LIN {X -0.033,Y -434.325,Z 655.091,A 0.000,B 0.000,C 90.000,E1 52.316} C_DIS
LIN {X -0.057,Y -434.303,Z 655.091,A 0.000,B 0.000,C 90.000,E1 52.316} C_DIS
LIN {X 0.127,Y -431.665,Z 655.083,A 0.000,B 0.000,C 90.000,E1 50.884} C_DIS
LIN {X 0.114,Y -427.591,Z 655.074,A 0.000,B 0.000,C 90.000,E1 49.218} C_DIS
LIN {X -0.216,Y -420.194,Z 655.054,A 0.000,B 0.000,C 90.000,E1 45.729} C_DIS
LIN {X -0.185,Y -420.290,Z 655.044,A 0.000,B 0.000,C 90.000,E1 44.028} C_DIS
LIN {X 0.050,Y -420.496,Z 655.033,A 0.000,B 0.000,C 90.000,E1 41.962} C_DIS
LIN {X 0.067,Y -421.322,Z 655.016,A 0.000,B 0.000,C 90.000,E1 38.910} C_DIS
LIN {X 0.145,Y -422.879,Z 654.997,A 0.000,B 0.000,C 90.000,E1 35.518} C_DIS
LIN {X 0.123,Y -423.713,Z 654.988,A 0.000,B 0.000,C 90.000,E1 33.833} C_DIS
LIN {X 0.233,Y -424.563,Z 654.979,A 0.000,B 0.000,C 90.000,E1 32.133} C_DIS
LIN {X 0.121,Y -425.591,Z 654.968,A 0.000,B 0.000,C 90.000,E1 30.129} C_DIS
LIN {X -0.166,Y -426.462,Z 654.958,A 0.000,B 0.000,C 90.000,E1 28.487} C_DIS
LIN {X 0.108,Y -427.566,Z 654.947,A 0.000,B 0.000,C 90.000,E1 26.437} C_DIS
LIN {X -0.129,Y -428.218,Z 654.941,A 0.000,B 0.000,C 90.000,E1 25.463} C_DIS
LIN {X 0.186,Y -430.765,Z 654.923,A 0.000,B 0.000,C 90.000,E1 22.078} C_DIS
LIN {X -0.161,Y -431.922,Z 654.915,A 0.000,B 0.000,C 90.000,E1 20.791} C_DIS
LIN {X -0.084,Y -432.910,Z 654.908,A 0.000,B 0.000,C 90.000,E1 19.450} C_DIS
LIN {X 0.100,Y -433.906,Z 654.899,A 0.000,B 0.000,C 90.000,E1 17.764} C_DIS
LIN {X -0.113,Y -434.974,Z 654.890,A 0.000,B 0.000,C 90.000,E1 16.134} C_DIS
LIN {X -0.194,Y -436.724,Z 654.877,A 0.000,B 0.000,C 90.000,E1 13.828} C_DIS
LIN {X -0.037,Y -438.454,Z 654.866,A 0.000,B 0.000,C 90.000,E1 11.827} C_DIS
LIN {X -0.141,Y -440.993,Z 654.851,A 0.000,B 0.000,C 90.000,E1 9.208} C_DIS
LIN {X 0.147,Y -443.830,Z 654.837,A 0.000,B 0.000,C 90.000,E1 6.549} C_DIS
LIN {X 0.026,Y -446.972,Z 654.822,A 0.000,B 0.000,C 90.000,E1 3.955} C_DIS
LIN {X 0.025,Y -449.568,Z 654.811,A 0.000,B 0.000,C 90.000,E1 2.007} C_DIS
LIN {X 0.058,Y -453.757,Z 654.795,A 0.000,B 0.000,C 90.000,E1 359.141} C_DIS
LIN {X 0.221,Y -456.932,Z 654.785,A 0.000,B 0.000,C 90.000,E1 357.192} C_DIS
LIN {X -0.208,Y -460.784,Z 654.772,A 0.000,B 0.000,C 90.000,E1 355.008} C_DIS
LIN {X 0.195,Y -463.089,Z 654.765,A 0.000,B 0.000,C 90.000,E1 353.685} C_DIS
LIN {X -0.239,Y -466.510,Z 654.755,A 0.000,B 0.000,C 90.000,E1 351.837} C_DIS
LIN {X 0.113,Y -469.285,Z 654.746,A 0.000,B 0.000,C 90.000,E1 350.218} C_DIS
LIN {X -0.153,Y -471.492,Z 654.739,A 0.000,B 0.000,C 90.000,E1 348.993} C_DIS
LIN {X -0.164,Y -474.778,Z 654.728,A 0.000,B 0.000,C 90.000,E1 347.117} C_DIS
LIN {X 0.015,Y -478.271,Z 654.718,A 0.000,B 0.000,C 90.000,E1 345.227} C_DIS
LIN {X 0.109,Y -480.603,Z 654.711,A 0.000,B 0.000,C 90.000,E1 343.976} C_DIS
LIN {X 0.084,Y -484.163,Z 654.701,A 0.000,B 0.000,C 90.000,E1 342.127} C_DIS
LIN {X -0.035,Y -487.158,Z 654.692,A 0.000,B 0.000,C 90.000,E1 340.604} C_DIS
LIN {X -0.094,Y -490.244,Z 654.684,A 0.000,B 0.000,C 90.000,E1 339.082} C_DIS
LIN {X 0.079,Y -493.203,Z 654.675,A 0.000,B 0.000,C 90.000,E1 337.539} C_DIS
LIN {X -0.199,Y -495.417,Z 654.669,A 0.000,B 0.000,C 90.000,E1 336.357} C_DIS
LIN {X 0.207,Y -497.465,Z 654.662,A 0.000,B 0.000,C 90.000,E1 335.101} C_DIS
LIN {X -0.139,Y -500.502,Z 654.652,A 0.000,B 0.000,C 90.000,E1 333.332} C_DIS
LIN {X -0.046,Y -504.909,Z 654.638,A 0.000,B 0.000,C 90.000,E1 330.923} C_DIS
LIN {X 0.206,Y -507.111,Z 654.633,A 0.000,B 0.000,C 90.000,E1 329.999} C_DIS
LIN {X 0.155,Y -509.021,Z 654.630,A 0.000,B 0.000,C 90.000,E1 329.410} C_DIS
LIN {X 0.046,Y -510.413,Z 654.629,A 0.000,B 0.000,C 90.000,E1 329.125} C_DIS
LIN {X 0.203,Y -513.157,Z 654.626,A 0.000,B 0.000,C 90.000,E1 328.663} C_DIS
LIN {X 0.021,Y -514.198,Z 654.625,A 0.000,B 0.000,C 90.000,E1 328.535} C_DIS
LIN {X 0.150,Y -515.794,Z 654.624,A 0.000,B 0.000,C 90.000,E1 328.329} C_DIS
LIN {X 0.072,Y -520.333,Z 654.622,A 0.000,B 0.000,C 90.000,E1 327.916} C_DIS
LIN {X -0.043,Y -524.730,Z 654.620,A 0.000,B 0.000,C 90.000,E1 327.533} C_DIS
LIN {X -0.043,Y -530.397,Z 654.617,A 0.000,B 0.000,C 90.000,E1 327.089} C_DIS
LIN {X 0.127,Y -537.887,Z 654.614,A 0.000,B 0.000,C 90.000,E1 326.501} C_DIS
LIN {X -0.157,Y -549.360,Z 654.609,A 0.000,B 0.000,C 90.000,E1 325.595} C_DIS
LIN {X -0.014,Y -554.965,Z 654.606,A 0.000,B 0.000,C 90.000,E1 325.102} C_DIS
LIN {X 0.066,Y -563.274,Z 654.602,A 0.000,B 0.000,C 90.000,E1 324.356} C_DIS
LIN {X 0.115,Y -572.552,Z 654.597,A 0.000,B 0.000,C 90.000,E1 323.497} C_DIS
LIN {X -0.045,Y -581.777,Z 654.592,A 0.000,B 0.000,C 90.000,E1 322.637} C_DIS
LIN {X 0.170,Y -590.747,Z 654.588,A 0.000,B 0.000,C 90.000,E1 321.743} C_DIS
LIN {X 0.239,Y -600.993,Z 654.582,A 0.000,B 0.000,C 90.000,E1 320.723} C_DIS
LIN {X -0.099,Y -606.973,Z 654.578,A 0.000,B 0.000,C 90.000,E1 320.114} C_DIS
LIN {X -0.086,Y -612.730,Z 654.575,A 0.000,B 0.000,C 90.000,E1 319.461} C_DIS
LIN {X 0.197,Y -614.929,Z 654.573,A 0.000,B 0.000,C 90.000,E1 319.175} C_DIS
LIN {X 0.155,Y -619.853,Z 654.570,A 0.000,B 0.000,C 90.000,E1 318.566} C_DIS
LIN {X -0.154,Y -623.691,Z 654.567,A 0.000,B 0.000,C 90.000,E1 318.081} C_DIS
LIN {X -0.226,Y -630.914,Z 654.561,A 0.000,B 0.000,C 90.000,E1 317.067} C_DIS
LIN {X 0.045,Y -633.534,Z 654.559,A 0.000,B 0.000,C 90.000,E1 316.662} C_DIS
LIN {X 0.106,Y -640.171,Z 654.554,A 0.000,B 0.000,C 90.000,E1 315.648} C_DIS
LIN {X 0.282,Y -645.772,Z 654.549,A 0.000,B 0.000,C 90.000,E1 314.757} C_DIS
LIN {X 0.019,Y -652.541,Z 654.543,A 0.000,B 0.000,C 90.000,E1 313.662} C_DIS
LIN {X -0.143,Y -658.239,Z 654.537,A 0.000,B 0.000,C 90.000,E1 312.690} C_DIS
LIN {X -0.214,Y -662.767,Z 654.532,A 0.000,B 0.000,C 90.000,E1 311.838} C_DIS
LIN {X -0.237,Y -667.097,Z 654.528,A 0.000,B 0.000,C 90.000,E1 310.987} C_DIS
LIN {X -0.180,Y -671.728,Z 654.522,A 0.000,B 0.000,C 90.000,E1 310.011} C_DIS
LIN {X -0.078,Y -674.785,Z 654.518,A 0.000,B 0.000,C 90.000,E1 309.277} C_DIS
LIN {X 0.060,Y -677.581,Z 654.514,A 0.000,B 0.000,C 90.000,E1 308.543} C_DIS
LIN {X 0.224,Y -680.153,Z 654.510,A 0.000,B 0.000,C 90.000,E1 307.810} C_DIS
LIN {X 0.023,Y -683.292,Z 654.505,A 0.000,B 0.000,C 90.000,E1 306.870} C_DIS
LIN {X -0.169,Y -685.471,Z 654.501,A 0.000,B 0.000,C 90.000,E1 306.171} C_DIS
LIN {X -0.118,Y -688.806,Z 654.494,A 0.000,B 0.000,C 90.000,E1 304.978} C_DIS
LIN {X 0.344,Y -691.293,Z 654.489,A 0.000,B 0.000,C 90.000,E1 303.992} C_DIS
LIN {X -0.129,Y -693.536,Z 654.484,A 0.000,B 0.000,C 90.000,E1 303.086} C_DIS
LIN {X 0.003,Y -695.668,Z 654.479,A 0.000,B 0.000,C 90.000,E1 302.133} C_DIS
LIN {X -0.204,Y -697.619,Z 654.473,A 0.000,B 0.000,C 90.000,E1 301.209} C_DIS
LIN {X -0.024,Y -699.348,Z 654.468,A 0.000,B 0.000,C 90.000,E1 300.256} C_DIS
LIN {X 0.086,Y -701.210,Z 654.462,A 0.000,B 0.000,C 90.000,E1 299.077} C_DIS
LIN {X 0.292,Y -702.183,Z 654.458,A 0.000,B 0.000,C 90.000,E1 298.359} C_DIS
LIN {X 0.122,Y -703.675,Z 654.451,A 0.000,B 0.000,C 90.000,E1 297.206} C_DIS
LIN {X 0.004,Y -704.754,Z 654.446,A 0.000,B 0.000,C 90.000,E1 296.283} C_DIS
LIN {X -0.076,Y -704.994,Z 654.442,A 0.000,B 0.000,C 90.000,E1 295.591} C_DIS
LIN {X -0.437,Y -704.321,Z 654.440,A 0.000,B 0.000,C 90.000,E1 295.155} C_DIS
LIN {X -0.151,Y -703.852,Z 654.438,A 0.000,B 0.000,C 90.000,E1 294.899} C_DIS
LIN {X -0.008,Y -703.310,Z 654.438,A 0.000,B 0.000,C 90.000,E1 294.771} C_DIS
LIN {X -0.376,Y -700.448,Z 654.435,A 0.000,B 0.000,C 90.000,E1 294.335} C_DIS
LIN {X -0.238,Y -699.553,Z 654.434,A 0.000,B 0.000,C 90.000,E1 294.207} C_DIS
LIN {X -0.103,Y -698.220,Z 654.434,A 0.000,B 0.000,C 90.000,E1 294.079} C_DIS
LIN {X -0.394,Y -694.498,Z 654.433,A 0.000,B 0.000,C 90.000,E1 293.898} C_DIS
LIN {X 0.118,Y -690.985,Z 654.432,A 0.000,B 0.000,C 90.000,E1 293.695} C_DIS
LIN {X -0.140,Y -689.032,Z 654.431,A 0.000,B 0.000,C 90.000,E1 293.643} C_DIS
LIN {X 0.050,Y -681.862,Z 654.430,A 0.000,B 0.000,C 90.000,E1 293.462} C_DIS
LIN {X -0.125,Y -679.782,Z 654.430,A 0.000,B 0.000,C 90.000,E1 293.439} C_DIS
LIN {X -0.175,Y -669.975,Z 654.430,A 0.000,B 0.000,C 90.000,E1 293.334} C_DIS
LIN {X -0.128,Y -662.993,Z 654.429,A 0.000,B 0.000,C 90.000,E1 293.259} C_DIS
LIN {X 0.325,Y -652.595,Z 654.428,A 0.000,B 0.000,C 90.000,E1 293.078} C_DIS
LIN {X -0.159,Y -642.877,Z 654.427,A 0.000,B 0.000,C 90.000,E1 292.950} C_DIS
LIN {X 0.122,Y -629.510,Z 654.426,A 0.000,B 0.000,C 90.000,E1 292.642} C_DIS
LIN {X -0.263,Y -616.266,Z 654.424,A 0.000,B 0.000,C 90.000,E1 292.333} C_DIS
LIN {X -0.196,Y -595.968,Z 654.421,A 0.000,B 0.000,C 90.000,E1 291.716} C_DIS
LIN {X -0.091,Y -578.430,Z 654.418,A 0.000,B 0.000,C 90.000,E1 291.153} C_DIS
LIN {X -0.036,Y -564.068,Z 654.415,A 0.000,B 0.000,C 90.000,E1 290.737} C_DIS
LIN {X 0.221,Y -561.514,Z 654.415,A 0.000,B 0.000,C 90.000,E1 290.610} C_DIS
LIN {X -0.242,Y -559.361,Z 654.414,A 0.000,B 0.000,C 90.000,E1 290.556} C_DIS
LIN {X 0.074,Y -556.501,Z 654.413,A 0.000,B 0.000,C 90.000,E1 290.355} C_DIS
LIN {X 0.019,Y -556.445,Z 654.413,A 0.000,B 0.000,C 90.000,E1 290.355} C_DIS
LIN {X 0.127,Y -555.648,Z 654.412,A 0.000,B 0.000,C 90.000,E1 290.194} C_DIS
LIN {X 0.000,Y -555.094,Z 654.409,A 0.000,B 0.000,C 90.000,E1 289.685} C_DIS
LIN {X 0.116,Y -554.826,Z 654.400,A 0.000,B 0.000,C 90.000,E1 288.000} C_DIS
LIN {X 0.228,Y -554.405,Z 654.391,A 0.000,B 0.000,C 90.000,E1 286.315} C_DIS
LIN {X -0.097,Y -553.844,Z 654.383,A 0.000,B 0.000,C 90.000,E1 284.954} C_DIS
LIN {X 0.110,Y -553.179,Z 654.375,A 0.000,B 0.000,C 90.000,E1 283.536} C_DIS
LIN {X 0.299,Y -552.403,Z 654.368,A 0.000,B 0.000,C 90.000,E1 282.119} C_DIS
LIN {X -0.061,Y -551.460,Z 654.357,A 0.000,B 0.000,C 90.000,E1 280.197} C_DIS
LIN {X -0.120,Y -551.001,Z 654.349,A 0.000,B 0.000,C 90.000,E1 278.803} C_DIS
LIN {X -0.016,Y -550.364,Z 654.336,A 0.000,B 0.000,C 90.000,E1 276.549} C_DIS
LIN {X -0.038,Y -549.996,Z 654.326,A 0.000,B 0.000,C 90.000,E1 274.588} C_DIS
LIN {X -0.219,Y -549.723,Z 654.316,A 0.000,B 0.000,C 90.000,E1 272.922} C_DIS
LIN {X 0.115,Y -549.183,Z 654.307,A 0.000,B 0.000,C 90.000,E1 271.203} C_DIS
LIN {X -0.173,Y -548.544,Z 654.299,A 0.000,B 0.000,C 90.000,E1 269.828} C_DIS
LIN {X 0.137,Y -547.639,Z 654.290,A 0.000,B 0.000,C 90.000,E1 268.108} C_DIS
LIN {X -0.158,Y -546.914,Z 654.282,A 0.000,B 0.000,C 90.000,E1 266.731} C_DIS
LIN {X 0.068,Y -546.038,Z 654.274,A 0.000,B 0.000,C 90.000,E1 265.298} C_DIS
LIN {X -0.178,Y -544.953,Z 654.266,A 0.000,B 0.000,C 90.000,E1 263.913} C_DIS
LIN {X 0.026,Y -543.929,Z 654.260,A 0.000,B 0.000,C 90.000,E1 262.761} C_DIS
LIN {X -0.255,Y -542.397,Z 654.252,A 0.000,B 0.000,C 90.000,E1 261.376} C_DIS
LIN {X -0.109,Y -539.644,Z 654.236,A 0.000,B 0.000,C 90.000,E1 258.522} C_DIS
LIN {X -0.029,Y -537.903,Z 654.225,A 0.000,B 0.000,C 90.000,E1 256.520} C_DIS
LIN {X -0.302,Y -536.949,Z 654.219,A 0.000,B 0.000,C 90.000,E1 255.408} C_DIS
LIN {X 0.198,Y -535.974,Z 654.212,A 0.000,B 0.000,C 90.000,E1 254.212} C_DIS
LIN {X -0.053,Y -533.985,Z 654.201,A 0.000,B 0.000,C 90.000,E1 252.236} C_DIS
LIN {X -0.103,Y -532.964,Z 654.195,A 0.000,B 0.000,C 90.000,E1 251.094} C_DIS
LIN {X 0.003,Y -531.661,Z 654.189,A 0.000,B 0.000,C 90.000,E1 249.934} C_DIS
LIN {X 0.093,Y -530.115,Z 654.182,A 0.000,B 0.000,C 90.000,E1 248.773} C_DIS
LIN {X 0.024,Y -527.580,Z 654.173,A 0.000,B 0.000,C 90.000,E1 247.050} C_DIS
LIN {X -0.241,Y -525.710,Z 654.166,A 0.000,B 0.000,C 90.000,E1 245.921} C_DIS
LIN {X 0.164,Y -523.592,Z 654.160,A 0.000,B 0.000,C 90.000,E1 244.717} C_DIS
LIN {X 0.215,Y -520.776,Z 654.152,A 0.000,B 0.000,C 90.000,E1 243.256} C_DIS
LIN {X -0.013,Y -517.758,Z 654.143,A 0.000,B 0.000,C 90.000,E1 241.820} C_DIS
LIN {X 0.160,Y -514.647,Z 654.135,A 0.000,B 0.000,C 90.000,E1 240.333} C_DIS
LIN {X 0.073,Y -511.274,Z 654.127,A 0.000,B 0.000,C 90.000,E1 238.869} C_DIS
LIN {X -0.181,Y -507.275,Z 654.117,A 0.000,B 0.000,C 90.000,E1 237.120} C_DIS
LIN {X 0.249,Y -504.480,Z 654.111,A 0.000,B 0.000,C 90.000,E1 235.881} C_DIS
LIN {X 0.103,Y -500.618,Z 654.102,A 0.000,B 0.000,C 90.000,E1 234.402} C_DIS
LIN {X -0.245,Y -495.933,Z 654.092,A 0.000,B 0.000,C 90.000,E1 232.637} C_DIS
LIN {X -0.095,Y -491.568,Z 654.082,A 0.000,B 0.000,C 90.000,E1 230.803} C_DIS
LIN {X 0.240,Y -485.807,Z 654.069,A 0.000,B 0.000,C 90.000,E1 228.324} C_DIS
LIN {X -0.065,Y -482.147,Z 654.060,A 0.000,B 0.000,C 90.000,E1 226.824} C_DIS
LIN {X 0.123,Y -479.203,Z 654.053,A 0.000,B 0.000,C 90.000,E1 225.567} C_DIS
LIN {X 0.140,Y -474.764,Z 654.043,A 0.000,B 0.000,C 90.000,E1 223.704} C_DIS
LIN {X -0.078,Y -469.069,Z 654.029,A 0.000,B 0.000,C 90.000,E1 221.229} C_DIS
LIN {X -0.174,Y -464.346,Z 654.017,A 0.000,B 0.000,C 90.000,E1 219.036} C_DIS
LIN {X -0.109,Y -461.027,Z 654.008,A 0.000,B 0.000,C 90.000,E1 217.443} C_DIS
LIN {X -0.003,Y -457.259,Z 653.997,A 0.000,B 0.000,C 90.000,E1 215.518} C_DIS
LIN {X 0.025,Y -454.278,Z 653.988,A 0.000,B 0.000,C 90.000,E1 213.913} C_DIS
LIN {X -0.082,Y -450.089,Z 653.976,A 0.000,B 0.000,C 90.000,E1 211.671} C_DIS
LIN {X -0.068,Y -447.168,Z 653.967,A 0.000,B 0.000,C 90.000,E1 210.050} C_DIS
LIN {X -0.016,Y -444.845,Z 653.960,A 0.000,B 0.000,C 90.000,E1 208.743} C_DIS
LIN {X -0.110,Y -441.283,Z 653.949,A 0.000,B 0.000,C 90.000,E1 206.796} C_DIS
LIN {X -0.095,Y -437.713,Z 653.938,A 0.000,B 0.000,C 90.000,E1 204.823} C_DIS
LIN {X 0.051,Y -434.722,Z 653.929,A 0.000,B 0.000,C 90.000,E1 203.153} C_DIS
LIN {X 0.125,Y -431.154,Z 653.918,A 0.000,B 0.000,C 90.000,E1 201.153} C_DIS
LIN {X -0.144,Y -427.095,Z 653.905,A 0.000,B 0.000,C 90.000,E1 198.852} C_DIS
LIN {X 0.103,Y -423.702,Z 653.893,A 0.000,B 0.000,C 90.000,E1 196.804} C_DIS
LIN {X 0.140,Y -420.426,Z 653.882,A 0.000,B 0.000,C 90.000,E1 194.773} C_DIS
LIN {X -0.115,Y -417.157,Z 653.871,A 0.000,B 0.000,C 90.000,E1 192.771} C_DIS
LIN {X 0.041,Y -412.955,Z 653.856,A 0.000,B 0.000,C 90.000,E1 190.018} C_DIS
LIN {X 0.191,Y -410.923,Z 653.848,A 0.000,B 0.000,C 90.000,E1 188.624} C_DIS
LIN {X -0.145,Y -407.386,Z 653.835,A 0.000,B 0.000,C 90.000,E1 186.258} C_DIS
LIN {X 0.144,Y -403.295,Z 653.817,A 0.000,B 0.000,C 90.000,E1 183.094} C_DIS
LIN {X -0.197,Y -399.883,Z 653.800,A 0.000,B 0.000,C 90.000,E1 180.000} C_DIS
LIN {X 0.169,Y -397.355,Z 653.782,A 0.000,B 0.000,C 90.000,E1 176.788} C_DIS
LIN {X 0.128,Y -395.783,Z 653.767,A 0.000,B 0.000,C 90.000,E1 173.976} C_DIS
LIN {X -0.122,Y -394.947,Z 653.755,A 0.000,B 0.000,C 90.000,E1 171.894} C_DIS
LIN {X -0.008,Y -394.356,Z 653.739,A 0.000,B 0.000,C 90.000,E1 169.050} C_DIS
LIN {X -0.112,Y -394.120,Z 653.721,A 0.000,B 0.000,C 90.000,E1 165.880} C_DIS
LIN {X 0.066,Y -394.291,Z 653.708,A 0.000,B 0.000,C 90.000,E1 163.378} C_DIS
LIN {X -0.012,Y -394.613,Z 653.694,A 0.000,B 0.000,C 90.000,E1 160.913} C_DIS
LIN {X -0.145,Y -394.848,Z 653.686,A 0.000,B 0.000,C 90.000,E1 159.518} C_DIS
LIN {X -0.183,Y -395.390,Z 653.672,A 0.000,B 0.000,C 90.000,E1 157.050} C_DIS
LIN {X 0.105,Y -395.907,Z 653.659,A 0.000,B 0.000,C 90.000,E1 154.537} C_DIS
LIN {X 0.178,Y -396.364,Z 653.647,A 0.000,B 0.000,C 90.000,E1 152.410} C_DIS
LIN {X -0.088,Y -396.937,Z 653.635,A 0.000,B 0.000,C 90.000,E1 150.333} C_DIS
LIN {X -0.079,Y -397.589,Z 653.621,A 0.000,B 0.000,C 90.000,E1 147.867} C_DIS
LIN {X 0.067,Y -398.195,Z 653.612,A 0.000,B 0.000,C 90.000,E1 146.087} C_DIS
LIN {X 0.104,Y -399.261,Z 653.598,A 0.000,B 0.000,C 90.000,E1 143.623} C_DIS
LIN {X -0.024,Y -400.225,Z 653.586,A 0.000,B 0.000,C 90.000,E1 141.537} C_DIS
LIN {X -0.079,Y -401.455,Z 653.573,A 0.000,B 0.000,C 90.000,E1 139.094} C_DIS
LIN {X 0.002,Y -402.564,Z 653.561,A 0.000,B 0.000,C 90.000,E1 136.986} C_DIS
LIN {X -0.006,Y -403.502,Z 653.551,A 0.000,B 0.000,C 90.000,E1 135.243} C_DIS
LIN {X -0.096,Y -405.540,Z 653.534,A 0.000,B 0.000,C 90.000,E1 132.123} C_DIS
LIN {X 0.089,Y -406.483,Z 653.529,A 0.000,B 0.000,C 90.000,E1 131.229} C_DIS
LIN {X 0.148,Y -407.602,Z 653.526,A 0.000,B 0.000,C 90.000,E1 130.701} C_DIS
LIN {X -0.018,Y -408.392,Z 653.524,A 0.000,B 0.000,C 90.000,E1 130.378} C_DIS
LIN {X 0.216,Y -409.094,Z 653.523,A 0.000,B 0.000,C 90.000,E1 130.172} C_DIS
LIN {X 0.059,Y -410.453,Z 653.521,A 0.000,B 0.000,C 90.000,E1 129.806} C_DIS
LIN {X -0.131,Y -413.741,Z 653.519,A 0.000,B 0.000,C 90.000,E1 129.358} C_DIS
LIN {X -0.118,Y -416.974,Z 653.517,A 0.000,B 0.000,C 90.000,E1 129.036} C_DIS
LIN {X -0.103,Y -421.967,Z 653.515,A 0.000,B 0.000,C 90.000,E1 128.624} C_DIS
LIN {X 0.194,Y -429.696,Z 653.511,A 0.000,B 0.000,C 90.000,E1 128.016} C_DIS
LIN {X 0.004,Y -436.340,Z 653.509,A 0.000,B 0.000,C 90.000,E1 127.569} C_DIS
LIN {X -0.075,Y -450.921,Z 653.503,A 0.000,B 0.000,C 90.000,E1 126.583} C_DIS
LIN {X -0.164,Y -462.119,Z 653.499,A 0.000,B 0.000,C 90.000,E1 125.804} C_DIS
LIN {X 0.120,Y -468.409,Z 653.496,A 0.000,B 0.000,C 90.000,E1 125.311} C_DIS
LIN {X -0.187,Y -480.823,Z 653.491,A 0.000,B 0.000,C 90.000,E1 124.405} C_DIS
LIN {X -0.091,Y -488.249,Z 653.488,A 0.000,B 0.000,C 90.000,E1 123.785} C_DIS
LIN {X 0.106,Y -496.820,Z 653.484,A 0.000,B 0.000,C 90.000,E1 123.038} C_DIS
LIN {X 0.079,Y -508.137,Z 653.478,A 0.000,B 0.000,C 90.000,E1 122.005} C_DIS
LIN {X -0.090,Y -514.962,Z 653.474,A 0.000,B 0.000,C 90.000,E1 121.386} C_DIS
LIN {X -0.114,Y -521.788,Z 653.471,A 0.000,B 0.000,C 90.000,E1 120.718} C_DIS
LIN {X 0.241,Y -526.990,Z 653.468,A 0.000,B 0.000,C 90.000,E1 120.129} C_DIS
LIN {X 0.090,Y -531.773,Z 653.465,A 0.000,B 0.000,C 90.000,E1 119.617} C_DIS
LIN {X 0.204,Y -536.168,Z 653.462,A 0.000,B 0.000,C 90.000,E1 119.077} C_DIS
LIN {X -0.125,Y -540.425,Z 653.459,A 0.000,B 0.000,C 90.000,E1 118.565} C_DIS
LIN {X -0.004,Y -544.201,Z 653.456,A 0.000,B 0.000,C 90.000,E1 118.025} C_DIS
LIN {X -0.154,Y -548.668,Z 653.452,A 0.000,B 0.000,C 90.000,E1 117.334} C_DIS
LIN {X -0.009,Y -552.514,Z 653.448,A 0.000,B 0.000,C 90.000,E1 116.616} C_DIS
LIN {X -0.074,Y -556.096,Z 653.444,A 0.000,B 0.000,C 90.000,E1 115.924} C_DIS
LIN {X 0.132,Y -559.198,Z 653.440,A 0.000,B 0.000,C 90.000,E1 115.207} C_DIS
LIN {X -0.180,Y -563.754,Z 653.434,A 0.000,B 0.000,C 90.000,E1 114.131} C_DIS
LIN {X 0.269,Y -566.998,Z 653.429,A 0.000,B 0.000,C 90.000,E1 113.259} C_DIS
LIN {X 0.015,Y -569.930,Z 653.425,A 0.000,B 0.000,C 90.000,E1 112.461} C_DIS
LIN {X 0.006,Y -572.587,Z 653.420,A 0.000,B 0.000,C 90.000,E1 111.642} C_DIS
LIN {X -0.193,Y -574.998,Z 653.416,A 0.000,B 0.000,C 90.000,E1 110.844} C_DIS
LIN {X 0.187,Y -578.411,Z 653.408,A 0.000,B 0.000,C 90.000,E1 109.450} C_DIS
LIN {X -0.140,Y -580.338,Z 653.404,A 0.000,B 0.000,C 90.000,E1 108.671} C_DIS
LIN {X -0.215,Y -583.227,Z 653.396,A 0.000,B 0.000,C 90.000,E1 107.330} C_DIS
LIN {X -0.197,Y -586.668,Z 653.387,A 0.000,B 0.000,C 90.000,E1 105.717} C_DIS
LIN {X 0.259,Y -591.327,Z 653.375,A 0.000,B 0.000,C 90.000,E1 103.536} C_DIS
LIN {X -0.116,Y -594.164,Z 653.368,A 0.000,B 0.000,C 90.000,E1 102.243} C_DIS
LIN {X 0.135,Y -596.935,Z 653.361,A 0.000,B 0.000,C 90.000,E1 100.894} C_DIS
LIN {X 0.029,Y -600.214,Z 653.352,A 0.000,B 0.000,C 90.000,E1 99.321} C_DIS
LIN {X 0.177,Y -602.813,Z 653.345,A 0.000,B 0.000,C 90.000,E1 97.992} C_DIS
LIN {X 0.139,Y -604.673,Z 653.339,A 0.000,B 0.000,C 90.000,E1 96.947} C_DIS
LIN {X 0.044,Y -606.484,Z 653.333,A 0.000,B 0.000,C 90.000,E1 95.910} C_DIS
LIN {X -0.107,Y -608.829,Z 653.324,A 0.000,B 0.000,C 90.000,E1 94.359} C_DIS
LIN {X 0.120,Y -610.679,Z 653.317,A 0.000,B 0.000,C 90.000,E1 93.037} C_DIS
LIN {X 0.014,Y -612.361,Z 653.308,A 0.000,B 0.000,C 90.000,E1 91.489} C_DIS
LIN {X -0.046,Y -613.252,Z 653.303,A 0.000,B 0.000,C 90.000,E1 90.458} C_DIS
LIN {X 0.227,Y -613.795,Z 653.298,A 0.000,B 0.000,C 90.000,E1 89.656} C_DIS
LIN {X 0.188,Y -614.324,Z 653.292,A 0.000,B 0.000,C 90.000,E1 88.625} C_DIS
LIN {X 0.170,Y -614.625,Z 653.287,A 0.000,B 0.000,C 90.000,E1 87.593} C_DIS
LIN {X -0.134,Y -614.758,Z 653.282,A 0.000,B 0.000,C 90.000,E1 86.846} C_DIS
LIN {X -0.138,Y -614.715,Z 653.277,A 0.000,B 0.000,C 90.000,E1 85.812} C_DIS
LIN {X 0.195,Y -614.350,Z 653.270,A 0.000,B 0.000,C 90.000,E1 84.489} C_DIS
LIN {X 0.167,Y -613.909,Z 653.264,A 0.000,B 0.000,C 90.000,E1 83.457} C_DIS
LIN {X 0.270,Y -613.340,Z 653.258,A 0.000,B 0.000,C 90.000,E1 82.413} C_DIS
LIN {X -0.319,Y -612.541,Z 653.252,A 0.000,B 0.000,C 90.000,E1 81.432} C_DIS
LIN {X -0.130,Y -610.777,Z 653.244,A 0.000,B 0.000,C 90.000,E1 79.859} C_DIS
LIN {X 0.282,Y -609.078,Z 653.236,A 0.000,B 0.000,C 90.000,E1 78.522} C_DIS
LIN {X 0.186,Y -607.161,Z 653.229,A 0.000,B 0.000,C 90.000,E1 77.229} C_DIS
LIN {X 0.058,Y -605.085,Z 653.222,A 0.000,B 0.000,C 90.000,E1 75.936} C_DIS
LIN {X 0.041,Y -602.779,Z 653.215,A 0.000,B 0.000,C 90.000,E1 74.629} C_DIS
LIN {X -0.017,Y -600.306,Z 653.207,A 0.000,B 0.000,C 90.000,E1 73.323} C_DIS
LIN {X 0.051,Y -597.637,Z 653.200,A 0.000,B 0.000,C 90.000,E1 72.000} C_DIS
LIN {X -0.189,Y -595.247,Z 653.194,A 0.000,B 0.000,C 90.000,E1 70.967} C_DIS
LIN {X 0.099,Y -592.668,Z 653.188,A 0.000,B 0.000,C 90.000,E1 69.880} C_DIS
LIN {X 0.111,Y -590.521,Z 653.184,A 0.000,B 0.000,C 90.000,E1 69.082} C_DIS
LIN {X 0.102,Y -588.176,Z 653.179,A 0.000,B 0.000,C 90.000,E1 68.284} C_DIS
LIN {X 0.066,Y -585.603,Z 653.175,A 0.000,B 0.000,C 90.000,E1 67.486} C_DIS
LIN {X -0.181,Y -583.795,Z 653.172,A 0.000,B 0.000,C 90.000,E1 66.975} C_DIS
LIN {X 0.129,Y -579.675,Z 653.166,A 0.000,B 0.000,C 90.000,E1 65.869} C_DIS
LIN {X 0.082,Y -575.434,Z 653.160,A 0.000,B 0.000,C 90.000,E1 64.793} C_DIS
LIN {X -0.221,Y -573.115,Z 653.157,A 0.000,B 0.000,C 90.000,E1 64.280} C_DIS
LIN {X 0.067,Y -569.505,Z 653.153,A 0.000,B 0.000,C 90.000,E1 63.435} C_DIS
LIN {X 0.051,Y -565.533,Z 653.148,A 0.000,B 0.000,C 90.000,E1 62.615} C_DIS
LIN {X -0.225,Y -563.352,Z 653.146,A 0.000,B 0.000,C 90.000,E1 62.231} C_DIS
LIN {X 0.150,Y -560.300,Z 653.143,A 0.000,B 0.000,C 90.000,E1 61.641} C_DIS
LIN {X 0.033,Y -556.114,Z 653.139,A 0.000,B 0.000,C 90.000,E1 60.973} C_DIS
LIN {X -0.252,Y -551.407,Z 653.135,A 0.000,B 0.000,C 90.000,E1 60.333} C_DIS
LIN {X -0.099,Y -547.510,Z 653.132,A 0.000,B 0.000,C 90.000,E1 59.793} C_DIS
LIN {X 0.156,Y -542.722,Z 653.129,A 0.000,B 0.000,C 90.000,E1 59.203} C_DIS
LIN {X 0.064,Y -537.484,Z 653.126,A 0.000,B 0.000,C 90.000,E1 58.663} C_DIS
LIN {X -0.043,Y -532.338,Z 653.123,A 0.000,B 0.000,C 90.000,E1 58.201} C_DIS
LIN {X -0.165,Y -528.302,Z 653.121,A 0.000,B 0.000,C 90.000,E1 57.867} C_DIS
LIN {X 0.048,Y -521.880,Z 653.119,A 0.000,B 0.000,C 90.000,E1 57.375} C_DIS
LIN {X 0.118,Y -517.021,Z 653.117,A 0.000,B 0.000,C 90.000,E1 57.041} C_DIS
LIN {X 0.238,Y -510.328,Z 653.115,A 0.000,B 0.000,C 90.000,E1 56.628} C_DIS
LIN {X -0.149,Y -503.595,Z 653.113,A 0.000,B 0.000,C 90.000,E1 56.294} C_DIS
LIN {X -0.111,Y -496.760,Z 653.111,A 0.000,B 0.000,C 90.000,E1 55.928} C_DIS
LIN {X 0.055,Y -476.690,Z 653.105,A 0.000,B 0.000,C 90.000,E1 54.848} C_DIS
LIN {X -0.035,Y -450.032,Z 653.097,A 0.000,B 0.000,C 90.000,E1 53.417} C_DIS
LIN {X 0.155,Y -435.467,Z 653.092,A 0.000,B 0.000,C 90.000,E1 52.557} C_DIS
LIN {X -0.154,Y -434.792,Z 653.092,A 0.000,B 0.000,C 90.000,E1 52.557} C_DIS
LIN {X -0.178,Y -434.753,Z 653.092,A 0.000,B 0.000,C 90.000,E1 52.557} C_DIS
LIN {X -0.037,Y -431.278,Z 653.082,A 0.000,B 0.000,C 90.000,E1 50.723} C_DIS
LIN {X -0.034,Y -422.090,Z 653.059,A 0.000,B 0.000,C 90.000,E1 46.701} C_DIS
LIN {X -0.237,Y -420.789,Z 653.056,A 0.000,B 0.000,C 90.000,E1 46.053} C_DIS
LIN {X 0.011,Y -420.605,Z 653.055,A 0.000,B 0.000,C 90.000,E1 45.850} C_DIS
LIN {X -0.179,Y -420.784,Z 653.046,A 0.000,B 0.000,C 90.000,E1 44.352} C_DIS
LIN {X 0.071,Y -420.990,Z 653.035,A 0.000,B 0.000,C 90.000,E1 42.285} C_DIS
LIN {X -0.214,Y -421.769,Z 653.018,A 0.000,B 0.000,C 90.000,E1 39.277} C_DIS
LIN {X 0.048,Y -422.906,Z 653.003,A 0.000,B 0.000,C 90.000,E1 36.537} C_DIS
LIN {X 0.100,Y -423.467,Z 652.997,A 0.000,B 0.000,C 90.000,E1 35.518} C_DIS
LIN {X -0.122,Y -424.148,Z 652.990,A 0.000,B 0.000,C 90.000,E1 34.199} C_DIS
LIN {X 0.211,Y -425.135,Z 652.979,A 0.000,B 0.000,C 90.000,E1 32.133} C_DIS
LIN {X 0.113,Y -426.134,Z 652.968,A 0.000,B 0.000,C 90.000,E1 30.129} C_DIS
LIN {X -0.165,Y -426.998,Z 652.958,A 0.000,B 0.000,C 90.000,E1 28.487} C_DIS
LIN {X 0.109,Y -428.328,Z 652.945,A 0.000,B 0.000,C 90.000,E1 26.104} C_DIS
LIN {X 0.041,Y -430.633,Z 652.927,A 0.000,B 0.000,C 90.000,E1 22.770} C_DIS
LIN {X 0.070,Y -432.079,Z 652.917,A 0.000,B 0.000,C 90.000,E1 21.099} C_DIS
LIN {X -0.031,Y -433.303,Z 652.908,A 0.000,B 0.000,C 90.000,E1 19.450} C_DIS
LIN {X -0.020,Y -434.482,Z 652.897,A 0.000,B 0.000,C 90.000,E1 17.457} C_DIS
LIN {X -0.115,Y -435.781,Z 652.886,A 0.000,B 0.000,C 90.000,E1 15.481} C_DIS
LIN {X -0.037,Y -437.903,Z 652.871,A 0.000,B 0.000,C 90.000,E1 12.827} C_DIS
LIN {X 0.057,Y -439.621,Z 652.860,A 0.000,B 0.000,C 90.000,E1 10.838} C_DIS
LIN {X 0.112,Y -441.575,Z 652.849,A 0.000,B 0.000,C 90.000,E1 8.859} C_DIS
LIN {X -0.189,Y -444.080,Z 652.837,A 0.000,B 0.000,C 90.000,E1 6.606} C_DIS
LIN {X -0.028,Y -446.747,Z 652.824,A 0.000,B 0.000,C 90.000,E1 4.302} C_DIS
LIN {X 0.143,Y -448.452,Z 652.817,A 0.000,B 0.000,C 90.000,E1 2.980} C_DIS
LIN {X 0.049,Y -452.022,Z 652.802,A 0.000,B 0.000,C 90.000,E1 0.401} C_DIS
LIN {X -0.135,Y -455.995,Z 652.788,A 0.000,B 0.000,C 90.000,E1 357.879} C_DIS
LIN {X -0.160,Y -459.789,Z 652.776,A 0.000,B 0.000,C 90.000,E1 355.641} C_DIS
LIN {X -0.038,Y -462.638,Z 652.767,A 0.000,B 0.000,C 90.000,E1 354.033} C_DIS
LIN {X 0.239,Y -465.457,Z 652.758,A 0.000,B 0.000,C 90.000,E1 352.413} C_DIS
LIN {X -0.153,Y -467.743,Z 652.751,A 0.000,B 0.000,C 90.000,E1 351.197} C_DIS
LIN {X 0.042,Y -471.058,Z 652.741,A 0.000,B 0.000,C 90.000,E1 349.285} C_DIS
LIN {X -0.145,Y -474.852,Z 652.728,A 0.000,B 0.000,C 90.000,E1 347.117} C_DIS
LIN {X -0.123,Y -478.951,Z 652.716,A 0.000,B 0.000,C 90.000,E1 344.936} C_DIS
LIN {X -0.190,Y -482.428,Z 652.706,A 0.000,B 0.000,C 90.000,E1 343.087} C_DIS
LIN {X -0.034,Y -486.043,Z 652.696,A 0.000,B 0.000,C 90.000,E1 341.221} C_DIS
LIN {X -0.067,Y -490.306,Z 652.684,A 0.000,B 0.000,C 90.000,E1 339.082} C_DIS
LIN {X 0.107,Y -493.257,Z 652.675,A 0.000,B 0.000,C 90.000,E1 337.539} C_DIS
LIN {X -0.171,Y -495.444,Z 652.669,A 0.000,B 0.000,C 90.000,E1 336.357} C_DIS
LIN {X 0.236,Y -497.488,Z 652.662,A 0.000,B 0.000,C 90.000,E1 335.101} C_DIS
LIN {X -0.110,Y -500.496,Z 652.652,A 0.000,B 0.000,C 90.000,E1 333.332} C_DIS
LIN {X 0.294,Y -505.432,Z 652.637,A 0.000,B 0.000,C 90.000,E1 330.589} C_DIS
LIN {X -0.141,Y -507.593,Z 652.632,A 0.000,B 0.000,C 90.000,E1 329.744} C_DIS
LIN {X 0.070,Y -509.547,Z 652.629,A 0.000,B 0.000,C 90.000,E1 329.125} C_DIS
LIN {X -0.014,Y -511.062,Z 652.627,A 0.000,B 0.000,C 90.000,E1 328.791} C_DIS
LIN {X -0.030,Y -513.017,Z 652.625,A 0.000,B 0.000,C 90.000,E1 328.456} C_DIS
LIN {X 0.044,Y -515.238,Z 652.623,A 0.000,B 0.000,C 90.000,E1 328.152} C_DIS
LIN {X 0.139,Y -516.431,Z 652.622,A 0.000,B 0.000,C 90.000,E1 327.995} C_DIS
LIN {X 0.064,Y -520.438,Z 652.620,A 0.000,B 0.000,C 90.000,E1 327.612} C_DIS
LIN {X -0.133,Y -525.746,Z 652.618,A 0.000,B 0.000,C 90.000,E1 327.168} C_DIS
LIN {X 0.026,Y -535.818,Z 652.613,A 0.000,B 0.000,C 90.000,E1 326.373} C_DIS
LIN {X -0.264,Y -547.461,Z 652.608,A 0.000,B 0.000,C 90.000,E1 325.468} C_DIS
LIN {X -0.090,Y -554.513,Z 652.605,A 0.000,B 0.000,C 90.000,E1 324.848} C_DIS
LIN {X -0.077,Y -562.894,Z 652.601,A 0.000,B 0.000,C 90.000,E1 324.116} C_DIS
LIN {X -0.067,Y -569.664,Z 652.597,A 0.000,B 0.000,C 90.000,E1 323.497} C_DIS
LIN {X 0.200,Y -580.237,Z 652.592,A 0.000,B 0.000,C 90.000,E1 322.477} C_DIS
LIN {X 0.064,Y -589.288,Z 652.587,A 0.000,B 0.000,C 90.000,E1 321.618} C_DIS
LIN {X -0.293,Y -600.894,Z 652.581,A 0.000,B 0.000,C 90.000,E1 320.517} C_DIS
LIN {X 0.201,Y -606.934,Z 652.577,A 0.000,B 0.000,C 90.000,E1 319.828} C_DIS
LIN {X -0.253,Y -612.740,Z 652.573,A 0.000,B 0.000,C 90.000,E1 319.218} C_DIS
LIN {X -0.202,Y -618.156,Z 652.570,A 0.000,B 0.000,C 90.000,E1 318.566} C_DIS
LIN {X -0.059,Y -622.125,Z 652.567,A 0.000,B 0.000,C 90.000,E1 318.038} C_DIS
LIN {X 0.270,Y -629.486,Z 652.561,A 0.000,B 0.000,C 90.000,E1 316.986} C_DIS
LIN {X 0.033,Y -632.998,Z 652.558,A 0.000,B 0.000,C 90.000,E1 316.500} C_DIS
LIN {X 0.085,Y -639.716,Z 652.553,A 0.000,B 0.000,C 90.000,E1 315.486} C_DIS
LIN {X 0.256,Y -645.340,Z 652.548,A 0.000,B 0.000,C 90.000,E1 314.595} C_DIS
LIN {X 0.194,Y -651.382,Z 652.542,A 0.000,B 0.000,C 90.000,E1 313.623} C_DIS
LIN {X -0.255,Y -657.147,Z 652.537,A 0.000,B 0.000,C 90.000,E1 312.690} C_DIS
LIN {X -0.339,Y -661.769,Z 652.532,A 0.000,B 0.000,C 90.000,E1 311.838} C_DIS
LIN {X 0.104,Y -665.633,Z 652.528,A 0.000,B 0.000,C 90.000,E1 311.067} C_DIS
LIN {X 0.145,Y -670.346,Z 652.523,A 0.000,B 0.000,C 90.000,E1 310.092} C_DIS
LIN {X 0.238,Y -673.570,Z 652.519,A 0.000,B 0.000,C 90.000,E1 309.358} C_DIS
LIN {X -0.164,Y -676.467,Z 652.515,A 0.000,B 0.000,C 90.000,E1 308.669} C_DIS
LIN {X -0.015,Y -679.113,Z 652.511,A 0.000,B 0.000,C 90.000,E1 307.935} C_DIS
LIN {X 0.311,Y -682.308,Z 652.505,A 0.000,B 0.000,C 90.000,E1 306.950} C_DIS
LIN {X 0.111,Y -684.558,Z 652.501,A 0.000,B 0.000,C 90.000,E1 306.251} C_DIS
LIN {X 0.177,Y -688.656,Z 652.494,A 0.000,B 0.000,C 90.000,E1 304.818} C_DIS
LIN {X -0.326,Y -691.141,Z 652.488,A 0.000,B 0.000,C 90.000,E1 303.913} C_DIS
LIN {X 0.003,Y -693.981,Z 652.482,A 0.000,B 0.000,C 90.000,E1 302.704} C_DIS
LIN {X -0.201,Y -696.621,Z 652.475,A 0.000,B 0.000,C 90.000,E1 301.544} C_DIS
LIN {X -0.032,Y -698.479,Z 652.470,A 0.000,B 0.000,C 90.000,E1 300.590} C_DIS
LIN {X -0.200,Y -700.127,Z 652.465,A 0.000,B 0.000,C 90.000,E1 299.667} C_DIS
LIN {X 0.267,Y -701.647,Z 652.460,A 0.000,B 0.000,C 90.000,E1 298.693} C_DIS
LIN {X 0.416,Y -703.232,Z 652.453,A 0.000,B 0.000,C 90.000,E1 297.513} C_DIS
LIN {X 0.263,Y -704.647,Z 652.447,A 0.000,B 0.000,C 90.000,E1 296.360} C_DIS
LIN {X -0.083,Y -704.861,Z 652.445,A 0.000,B 0.000,C 90.000,E1 296.155} C_DIS
LIN {X 0.185,Y -704.999,Z 652.443,A 0.000,B 0.000,C 90.000,E1 295.668} C_DIS
LIN {X -0.162,Y -704.829,Z 652.441,A 0.000,B 0.000,C 90.000,E1 295.463} C_DIS
LIN {X 0.114,Y -704.106,Z 652.439,A 0.000,B 0.000,C 90.000,E1 294.975} C_DIS
LIN {X -0.238,Y -703.189,Z 652.438,A 0.000,B 0.000,C 90.000,E1 294.771} C_DIS
LIN {X 0.321,Y -700.318,Z 652.435,A 0.000,B 0.000,C 90.000,E1 294.259} C_DIS
LIN {X 0.171,Y -699.364,Z 652.434,A 0.000,B 0.000,C 90.000,E1 294.155} C_DIS
LIN {X -0.332,Y -697.936,Z 652.434,A 0.000,B 0.000,C 90.000,E1 294.079} C_DIS
LIN {X -0.074,Y -695.897,Z 652.433,A 0.000,B 0.000,C 90.000,E1 293.951} C_DIS
LIN {X -0.044,Y -690.251,Z 652.432,A 0.000,B 0.000,C 90.000,E1 293.695} C_DIS
LIN {X -0.262,Y -688.188,Z 652.431,A 0.000,B 0.000,C 90.000,E1 293.643} C_DIS
LIN {X 0.088,Y -681.443,Z 652.430,A 0.000,B 0.000,C 90.000,E1 293.462} C_DIS
LIN {X -0.217,Y -673.441,Z 652.430,A 0.000,B 0.000,C 90.000,E1 293.387} C_DIS
LIN {X 0.131,Y -663.519,Z 652.429,A 0.000,B 0.000,C 90.000,E1 293.259} C_DIS
LIN {X 0.078,Y -653.615,Z 652.429,A 0.000,B 0.000,C 90.000,E1 293.131} C_DIS
LIN {X 0.221,Y -643.660,Z 652.428,A 0.000,B 0.000,C 90.000,E1 292.950} C_DIS
LIN {X -0.046,Y -630.294,Z 652.426,A 0.000,B 0.000,C 90.000,E1 292.695} C_DIS
LIN {X -0.212,Y -620.523,Z 652.425,A 0.000,B 0.000,C 90.000,E1 292.461} C_DIS
LIN {X -0.185,Y -603.676,Z 652.422,A 0.000,B 0.000,C 90.000,E1 291.972} C_DIS
LIN {X 0.135,Y -582.740,Z 652.418,A 0.000,B 0.000,C 90.000,E1 291.280} C_DIS
LIN {X -0.243,Y -575.451,Z 652.417,A 0.000,B 0.000,C 90.000,E1 291.099} C_DIS
LIN {X -0.109,Y -563.481,Z 652.415,A 0.000,B 0.000,C 90.000,E1 290.737} C_DIS
LIN {X -0.062,Y -560.523,Z 652.414,A 0.000,B 0.000,C 90.000,E1 290.610} C_DIS
LIN {X 0.009,Y -556.596,Z 652.413,A 0.000,B 0.000,C 90.000,E1 290.375} C_DIS
LIN {X -0.047,Y -556.537,Z 652.413,A 0.000,B 0.000,C 90.000,E1 290.375} C_DIS
LIN {X -0.322,Y -555.710,Z 652.412,A 0.000,B 0.000,C 90.000,E1 290.248} C_DIS
LIN {X 0.073,Y -555.187,Z 652.409,A 0.000,B 0.000,C 90.000,E1 289.685} C_DIS
LIN {X 0.191,Y -554.933,Z 652.400,A 0.000,B 0.000,C 90.000,E1 288.000} C_DIS
LIN {X 0.305,Y -554.500,Z 652.391,A 0.000,B 0.000,C 90.000,E1 286.315} C_DIS
LIN {X -0.018,Y -553.954,Z 652.383,A 0.000,B 0.000,C 90.000,E1 284.954} C_DIS
LIN {X 0.192,Y -553.290,Z 652.375,A 0.000,B 0.000,C 90.000,E1 283.536} C_DIS
LIN {X -0.039,Y -552.366,Z 652.366,A 0.000,B 0.000,C 90.000,E1 281.883} C_DIS
LIN {X -0.173,Y -551.287,Z 652.352,A 0.000,B 0.000,C 90.000,E1 279.378} C_DIS
LIN {X -0.071,Y -550.605,Z 652.340,A 0.000,B 0.000,C 90.000,E1 277.125} C_DIS
LIN {X -0.131,Y -550.203,Z 652.330,A 0.000,B 0.000,C 90.000,E1 275.448} C_DIS
LIN {X 0.191,Y -549.961,Z 652.322,A 0.000,B 0.000,C 90.000,E1 274.012} C_DIS
LIN {X -0.125,Y -549.758,Z 652.316,A 0.000,B 0.000,C 90.000,E1 272.922} C_DIS
LIN {X 0.207,Y -549.245,Z 652.307,A 0.000,B 0.000,C 90.000,E1 271.203} C_DIS
LIN {X -0.079,Y -548.604,Z 652.299,A 0.000,B 0.000,C 90.000,E1 269.828} C_DIS
LIN {X -0.267,Y -547.573,Z 652.288,A 0.000,B 0.000,C 90.000,E1 267.879} C_DIS
LIN {X -0.020,Y -546.827,Z 652.280,A 0.000,B 0.000,C 90.000,E1 266.445} C_DIS
LIN {X 0.166,Y -546.139,Z 652.274,A 0.000,B 0.000,C 90.000,E1 265.298} C_DIS
LIN {X -0.078,Y -545.065,Z 652.266,A 0.000,B 0.000,C 90.000,E1 263.913} C_DIS
LIN {X 0.127,Y -544.061,Z 652.260,A 0.000,B 0.000,C 90.000,E1 262.761} C_DIS
LIN {X -0.152,Y -542.517,Z 652.252,A 0.000,B 0.000,C 90.000,E1 261.376} C_DIS
LIN {X -0.003,Y -539.761,Z 652.236,A 0.000,B 0.000,C 90.000,E1 258.522} C_DIS
LIN {X 0.145,Y -537.784,Z 652.224,A 0.000,B 0.000,C 90.000,E1 256.228} C_DIS
LIN {X 0.112,Y -536.346,Z 652.214,A 0.000,B 0.000,C 90.000,E1 254.519} C_DIS
LIN {X 0.092,Y -535.199,Z 652.208,A 0.000,B 0.000,C 90.000,E1 253.378} C_DIS
LIN {X -0.186,Y -533.321,Z 652.197,A 0.000,B 0.000,C 90.000,E1 251.402} C_DIS
LIN {X -0.272,Y -532.461,Z 652.192,A 0.000,B 0.000,C 90.000,E1 250.550} C_DIS
LIN {X -0.174,Y -531.038,Z 652.185,A 0.000,B 0.000,C 90.000,E1 249.390} C_DIS
LIN {X 0.086,Y -528.943,Z 652.177,A 0.000,B 0.000,C 90.000,E1 247.922} C_DIS
LIN {X 0.144,Y -527.681,Z 652.173,A 0.000,B 0.000,C 90.000,E1 247.050} C_DIS
LIN {X -0.120,Y -525.795,Z 652.166,A 0.000,B 0.000,C 90.000,E1 245.921} C_DIS
LIN {X 0.286,Y -523.672,Z 652.160,A 0.000,B 0.000,C 90.000,E1 244.717} C_DIS
LIN {X -0.127,Y -520.824,Z 652.152,A 0.000,B 0.000,C 90.000,E1 243.307} C_DIS
LIN {X -0.134,Y -517.792,Z 652.144,A 0.000,B 0.000,C 90.000,E1 241.847} C_DIS
LIN {X -0.078,Y -515.358,Z 652.137,A 0.000,B 0.000,C 90.000,E1 240.667} C_DIS
LIN {X -0.151,Y -511.976,Z 652.129,A 0.000,B 0.000,C 90.000,E1 239.203} C_DIS
LIN {X -0.016,Y -508.633,Z 652.121,A 0.000,B 0.000,C 90.000,E1 237.709} C_DIS
LIN {X 0.161,Y -505.874,Z 652.114,A 0.000,B 0.000,C 90.000,E1 236.501} C_DIS
LIN {X -0.048,Y -504.479,Z 652.111,A 0.000,B 0.000,C 90.000,E1 235.928} C_DIS
LIN {X -0.070,Y -501.373,Z 652.104,A 0.000,B 0.000,C 90.000,E1 234.736} C_DIS
LIN {X 0.006,Y -496.681,Z 652.094,A 0.000,B 0.000,C 90.000,E1 232.924} C_DIS
LIN {X 0.022,Y -491.547,Z 652.082,A 0.000,B 0.000,C 90.000,E1 230.803} C_DIS
LIN {X -0.009,Y -485.762,Z 652.069,A 0.000,B 0.000,C 90.000,E1 228.366} C_DIS
LIN {X 0.048,Y -482.108,Z 652.060,A 0.000,B 0.000,C 90.000,E1 226.824} C_DIS
LIN {X 0.234,Y -479.134,Z 652.053,A 0.000,B 0.000,C 90.000,E1 225.567} C_DIS
LIN {X 0.142,Y -475.465,Z 652.045,A 0.000,B 0.000,C 90.000,E1 224.028} C_DIS
LIN {X -0.052,Y -469.723,Z 652.031,A 0.000,B 0.000,C 90.000,E1 221.553} C_DIS
LIN {X -0.070,Y -464.270,Z 652.017,A 0.000,B 0.000,C 90.000,E1 219.036} C_DIS
LIN {X -0.260,Y -460.308,Z 652.006,A 0.000,B 0.000,C 90.000,E1 217.156} C_DIS
LIN {X -0.171,Y -456.556,Z 651.996,A 0.000,B 0.000,C 90.000,E1 215.231} C_DIS
LIN {X 0.220,Y -453.578,Z 651.987,A 0.000,B 0.000,C 90.000,E1 213.579} C_DIS
LIN {X 0.097,Y -449.467,Z 651.974,A 0.000,B 0.000,C 90.000,E1 211.337} C_DIS
LIN {X 0.012,Y -445.446,Z 651.962,A 0.000,B 0.000,C 90.000,E1 209.077} C_DIS
LIN {X -0.064,Y -441.841,Z 651.951,A 0.000,B 0.000,C 90.000,E1 207.129} C_DIS
LIN {X -0.029,Y -438.280,Z 651.940,A 0.000,B 0.000,C 90.000,E1 205.155} C_DIS
LIN {X 0.138,Y -434.657,Z 651.929,A 0.000,B 0.000,C 90.000,E1 203.153} C_DIS
LIN {X 0.055,Y -431.112,Z 651.918,A 0.000,B 0.000,C 90.000,E1 201.173} C_DIS
LIN {X -0.128,Y -427.633,Z 651.907,A 0.000,B 0.000,C 90.000,E1 199.195} C_DIS
LIN {X -0.005,Y -424.245,Z 651.895,A 0.000,B 0.000,C 90.000,E1 197.166} C_DIS
LIN {X 0.222,Y -420.410,Z 651.882,A 0.000,B 0.000,C 90.000,E1 194.773} C_DIS
LIN {X -0.034,Y -417.165,Z 651.871,A 0.000,B 0.000,C 90.000,E1 192.771} C_DIS
LIN {X 0.122,Y -412.978,Z 651.856,A 0.000,B 0.000,C 90.000,E1 190.018} C_DIS
LIN {X -0.135,Y -410.952,Z 651.848,A 0.000,B 0.000,C 90.000,E1 188.681} C_DIS
LIN {X -0.065,Y -407.420,Z 651.835,A 0.000,B 0.000,C 90.000,E1 186.258} C_DIS
LIN {X -0.177,Y -403.340,Z 651.817,A 0.000,B 0.000,C 90.000,E1 183.151} C_DIS
LIN {X -0.114,Y -399.937,Z 651.800,A 0.000,B 0.000,C 90.000,E1 180.000} C_DIS
LIN {X -0.107,Y -397.668,Z 651.784,A 0.000,B 0.000,C 90.000,E1 177.192} C_DIS
LIN {X -0.179,Y -395.869,Z 651.767,A 0.000,B 0.000,C 90.000,E1 174.033} C_DIS
LIN {X -0.034,Y -395.047,Z 651.755,A 0.000,B 0.000,C 90.000,E1 171.894} C_DIS
LIN {X 0.120,Y -394.518,Z 651.741,A 0.000,B 0.000,C 90.000,E1 169.398} C_DIS
LIN {X -0.022,Y -394.264,Z 651.726,A 0.000,B 0.000,C 90.000,E1 166.589} C_DIS
LIN {X 0.102,Y -394.317,Z 651.714,A 0.000,B 0.000,C 90.000,E1 164.448} C_DIS
LIN {X -0.207,Y -394.502,Z 651.704,A 0.000,B 0.000,C 90.000,E1 162.725} C_DIS
LIN {X 0.155,Y -394.850,Z 651.692,A 0.000,B 0.000,C 90.000,E1 160.550} C_DIS
LIN {X 0.225,Y -395.147,Z 651.682,A 0.000,B 0.000,C 90.000,E1 158.773} C_DIS
LIN {X -0.068,Y -395.578,Z 651.672,A 0.000,B 0.000,C 90.000,E1 157.050} C_DIS
LIN {X 0.087,Y -396.221,Z 651.657,A 0.000,B 0.000,C 90.000,E1 154.204} C_DIS
LIN {X -0.012,Y -396.695,Z 651.645,A 0.000,B 0.000,C 90.000,E1 152.103} C_DIS
LIN {X -0.082,Y -397.226,Z 651.633,A 0.000,B 0.000,C 90.000,E1 149.999} C_DIS
LIN {X 0.060,Y -397.811,Z 651.622,A 0.000,B 0.000,C 90.000,E1 147.867} C_DIS
LIN {X -0.121,Y -398.429,Z 651.612,A 0.000,B 0.000,C 90.000,E1 146.135} C_DIS
LIN {X 0.017,Y -399.462,Z 651.598,A 0.000,B 0.000,C 90.000,E1 143.657} C_DIS
LIN {X 0.016,Y -400.282,Z 651.588,A 0.000,B 0.000,C 90.000,E1 141.904} C_DIS
LIN {X -0.155,Y -401.263,Z 651.577,A 0.000,B 0.000,C 90.000,E1 139.828} C_DIS
LIN {X -0.164,Y -402.146,Z 651.567,A 0.000,B 0.000,C 90.000,E1 138.081} C_DIS
LIN {X -0.063,Y -403.227,Z 651.555,A 0.000,B 0.000,C 90.000,E1 135.972} C_DIS
LIN {X 0.222,Y -404.134,Z 651.546,A 0.000,B 0.000,C 90.000,E1 134.190} C_DIS
LIN {X 0.207,Y -405.776,Z 651.532,A 0.000,B 0.000,C 90.000,E1 131.757} C_DIS
LIN {X 0.176,Y -406.547,Z 651.528,A 0.000,B 0.000,C 90.000,E1 131.067} C_DIS
LIN {X 0.150,Y -407.789,Z 651.524,A 0.000,B 0.000,C 90.000,E1 130.378} C_DIS
LIN {X -0.060,Y -409.732,Z 651.521,A 0.000,B 0.000,C 90.000,E1 129.769} C_DIS
LIN {X 0.158,Y -411.311,Z 651.520,A 0.000,B 0.000,C 90.000,E1 129.483} C_DIS
LIN {X -0.183,Y -412.205,Z 651.519,A 0.000,B 0.000,C 90.000,E1 129.358} C_DIS
LIN {X 0.059,Y -413.369,Z 651.518,A 0.000,B 0.000,C 90.000,E1 129.152} C_DIS
LIN {X 0.017,Y -417.503,Z 651.515,A 0.000,B 0.000,C 90.000,E1 128.749} C_DIS
LIN {X -0.151,Y -422.309,Z 651.513,A 0.000,B 0.000,C 90.000,E1 128.382} C_DIS
LIN {X 0.212,Y -433.567,Z 651.509,A 0.000,B 0.000,C 90.000,E1 127.523} C_DIS
LIN {X 0.022,Y -449.811,Z 651.503,A 0.000,B 0.000,C 90.000,E1 126.457} C_DIS
LIN {X -0.098,Y -459.428,Z 651.499,A 0.000,B 0.000,C 90.000,E1 125.804} C_DIS
LIN {X 0.234,Y -465.730,Z 651.496,A 0.000,B 0.000,C 90.000,E1 125.311} C_DIS
LIN {X 0.085,Y -476.451,Z 651.492,A 0.000,B 0.000,C 90.000,E1 124.532} C_DIS
LIN {X 0.030,Y -482.491,Z 651.489,A 0.000,B 0.000,C 90.000,E1 124.072} C_DIS
LIN {X 0.187,Y -486.802,Z 651.487,A 0.000,B 0.000,C 90.000,E1 123.706} C_DIS
LIN {X 0.060,Y -495.422,Z 651.483,A 0.000,B 0.000,C 90.000,E1 123.007} C_DIS
LIN {X -0.100,Y -503.926,Z 651.479,A 0.000,B 0.000,C 90.000,E1 122.260} C_DIS
LIN {X -0.083,Y -512.113,Z 651.475,A 0.000,B 0.000,C 90.000,E1 121.514} C_DIS
LIN {X -0.139,Y -520.548,Z 651.471,A 0.000,B 0.000,C 90.000,E1 120.718} C_DIS
LIN {X -0.047,Y -526.812,Z 651.467,A 0.000,B 0.000,C 90.000,E1 120.050} C_DIS
LIN {X -0.009,Y -530.449,Z 651.465,A 0.000,B 0.000,C 90.000,E1 119.667} C_DIS
LIN {X -0.018,Y -534.889,Z 651.462,A 0.000,B 0.000,C 90.000,E1 119.155} C_DIS
LIN {X -0.071,Y -539.283,Z 651.459,A 0.000,B 0.000,C 90.000,E1 118.615} C_DIS
LIN {X -0.316,Y -544.182,Z 651.455,A 0.000,B 0.000,C 90.000,E1 117.975} C_DIS
LIN {X -0.090,Y -547.897,Z 651.452,A 0.000,B 0.000,C 90.000,E1 117.385} C_DIS
LIN {X -0.070,Y -552.629,Z 651.447,A 0.000,B 0.000,C 90.000,E1 116.539} C_DIS
LIN {X -0.139,Y -556.253,Z 651.444,A 0.000,B 0.000,C 90.000,E1 115.848} C_DIS
LIN {X -0.276,Y -559.975,Z 651.439,A 0.000,B 0.000,C 90.000,E1 115.027} C_DIS
LIN {X -0.062,Y -564.543,Z 651.433,A 0.000,B 0.000,C 90.000,E1 113.898} C_DIS
LIN {X -0.119,Y -567.799,Z 651.428,A 0.000,B 0.000,C 90.000,E1 113.078} C_DIS
LIN {X -0.149,Y -570.709,Z 651.424,A 0.000,B 0.000,C 90.000,E1 112.259} C_DIS
LIN {X 0.166,Y -573.327,Z 651.419,A 0.000,B 0.000,C 90.000,E1 111.408} C_DIS
LIN {X 0.150,Y -574.952,Z 651.416,A 0.000,B 0.000,C 90.000,E1 110.865} C_DIS
LIN {X -0.185,Y -577.820,Z 651.410,A 0.000,B 0.000,C 90.000,E1 109.812} C_DIS
LIN {X -0.136,Y -580.461,Z 651.404,A 0.000,B 0.000,C 90.000,E1 108.725} C_DIS
LIN {X 0.170,Y -583.387,Z 651.397,A 0.000,B 0.000,C 90.000,E1 107.347} C_DIS
LIN {X 0.044,Y -587.429,Z 651.386,A 0.000,B 0.000,C 90.000,E1 105.481} C_DIS
LIN {X 0.260,Y -591.574,Z 651.376,A 0.000,B 0.000,C 90.000,E1 103.592} C_DIS
LIN {X -0.113,Y -594.473,Z 651.368,A 0.000,B 0.000,C 90.000,E1 102.299} C_DIS
LIN {X -0.155,Y -597.832,Z 651.359,A 0.000,B 0.000,C 90.000,E1 100.715} C_DIS
LIN {X 0.039,Y -600.610,Z 651.352,A 0.000,B 0.000,C 90.000,E1 99.378} C_DIS
LIN {X 0.193,Y -603.264,Z 651.345,A 0.000,B 0.000,C 90.000,E1 98.049} C_DIS
LIN {X 0.159,Y -605.185,Z 651.339,A 0.000,B 0.000,C 90.000,E1 97.004} C_DIS
LIN {X -0.281,Y -607.412,Z 651.332,A 0.000,B 0.000,C 90.000,E1 95.739} C_DIS
LIN {X 0.199,Y -609.773,Z 651.323,A 0.000,B 0.000,C 90.000,E1 94.131} C_DIS
LIN {X 0.164,Y -611.242,Z 651.317,A 0.000,B 0.000,C 90.000,E1 93.094} C_DIS
LIN {X -0.239,Y -612.711,Z 651.310,A 0.000,B 0.000,C 90.000,E1 91.835} C_DIS
LIN {X 0.041,Y -613.471,Z 651.306,A 0.000,B 0.000,C 90.000,E1 91.031} C_DIS
LIN {X 0.298,Y -614.468,Z 651.299,A 0.000,B 0.000,C 90.000,E1 89.714} C_DIS
LIN {X 0.267,Y -614.995,Z 651.293,A 0.000,B 0.000,C 90.000,E1 88.682} C_DIS
LIN {X 0.260,Y -615.336,Z 651.287,A 0.000,B 0.000,C 90.000,E1 87.650} C_DIS
LIN {X 0.263,Y -615.461,Z 651.281,A 0.000,B 0.000,C 90.000,E1 86.617} C_DIS
LIN {X -0.055,Y -615.297,Z 651.274,A 0.000,B 0.000,C 90.000,E1 85.355} C_DIS
LIN {X 0.277,Y -614.829,Z 651.267,A 0.000,B 0.000,C 90.000,E1 84.033} C_DIS
LIN {X -0.294,Y -614.326,Z 651.261,A 0.000,B 0.000,C 90.000,E1 83.053} C_DIS
LIN {X -0.180,Y -613.638,Z 651.256,A 0.000,B 0.000,C 90.000,E1 82.008} C_DIS
LIN {X 0.185,Y -612.901,Z 651.251,A 0.000,B 0.000,C 90.000,E1 81.197} C_DIS
LIN {X -0.071,Y -611.408,Z 651.244,A 0.000,B 0.000,C 90.000,E1 79.926} C_DIS
LIN {X -0.136,Y -609.649,Z 651.237,A 0.000,B 0.000,C 90.000,E1 78.634} C_DIS
LIN {X 0.244,Y -607.742,Z 651.230,A 0.000,B 0.000,C 90.000,E1 77.297} C_DIS
LIN {X 0.262,Y -605.608,Z 651.222,A 0.000,B 0.000,C 90.000,E1 75.992} C_DIS
LIN {X -0.215,Y -603.744,Z 651.217,A 0.000,B 0.000,C 90.000,E1 74.991} C_DIS
LIN {X 0.019,Y -601.772,Z 651.211,A 0.000,B 0.000,C 90.000,E1 73.921} C_DIS
LIN {X 0.220,Y -599.680,Z 651.205,A 0.000,B 0.000,C 90.000,E1 72.851} C_DIS
LIN {X -0.002,Y -597.469,Z 651.199,A 0.000,B 0.000,C 90.000,E1 71.819} C_DIS
LIN {X -0.137,Y -595.660,Z 651.195,A 0.000,B 0.000,C 90.000,E1 71.040} C_DIS
LIN {X 0.353,Y -593.046,Z 651.189,A 0.000,B 0.000,C 90.000,E1 69.934} C_DIS
LIN {X 0.048,Y -590.058,Z 651.183,A 0.000,B 0.000,C 90.000,E1 68.901} C_DIS
LIN {X 0.032,Y -587.630,Z 651.178,A 0.000,B 0.000,C 90.000,E1 68.103} C_DIS
LIN {X -0.136,Y -583.990,Z 651.172,A 0.000,B 0.000,C 90.000,E1 67.050} C_DIS
LIN {X -0.122,Y -579.851,Z 651.167,A 0.000,B 0.000,C 90.000,E1 65.973} C_DIS
LIN {X -0.156,Y -575.539,Z 651.161,A 0.000,B 0.000,C 90.000,E1 64.897} C_DIS
LIN {X 0.064,Y -573.221,Z 651.157,A 0.000,B 0.000,C 90.000,E1 64.332} C_DIS
LIN {X 0.099,Y -569.505,Z 651.153,A 0.000,B 0.000,C 90.000,E1 63.512} C_DIS
LIN {X -0.244,Y -566.880,Z 651.150,A 0.000,B 0.000,C 90.000,E1 62.999} C_DIS
LIN {X 0.065,Y -563.299,Z 651.146,A 0.000,B 0.000,C 90.000,E1 62.281} C_DIS
LIN {X 0.076,Y -559.277,Z 651.142,A 0.000,B 0.000,C 90.000,E1 61.591} C_DIS
LIN {X -0.070,Y -555.792,Z 651.139,A 0.000,B 0.000,C 90.000,E1 61.051} C_DIS
LIN {X 0.139,Y -550.756,Z 651.135,A 0.000,B 0.000,C 90.000,E1 60.333} C_DIS
LIN {X 0.069,Y -547.557,Z 651.133,A 0.000,B 0.000,C 90.000,E1 59.921} C_DIS
LIN {X 0.329,Y -542.765,Z 651.130,A 0.000,B 0.000,C 90.000,E1 59.331} C_DIS
LIN {X -0.039,Y -537.465,Z 651.127,A 0.000,B 0.000,C 90.000,E1 58.820} C_DIS
LIN {X 0.007,Y -534.213,Z 651.125,A 0.000,B 0.000,C 90.000,E1 58.535} C_DIS
LIN {X 0.071,Y -532.076,Z 651.124,A 0.000,B 0.000,C 90.000,E1 58.329} C_DIS
LIN {X -0.062,Y -526.238,Z 651.122,A 0.000,B 0.000,C 90.000,E1 57.867} C_DIS
LIN {X 0.069,Y -521.278,Z 651.120,A 0.000,B 0.000,C 90.000,E1 57.502} C_DIS
LIN {X -0.240,Y -514.793,Z 651.117,A 0.000,B 0.000,C 90.000,E1 57.120} C_DIS
LIN {X -0.052,Y -507.965,Z 651.115,A 0.000,B 0.000,C 90.000,E1 56.707} C_DIS
LIN {X 0.297,Y -499.647,Z 651.113,A 0.000,B 0.000,C 90.000,E1 56.215} C_DIS
LIN {X 0.141,Y -479.576,Z 651.107,A 0.000,B 0.000,C 90.000,E1 55.182} C_DIS
LIN {X -0.138,Y -462.730,Z 651.102,A 0.000,B 0.000,C 90.000,E1 54.322} C_DIS
LIN {X 0.075,Y -444.555,Z 651.096,A 0.000,B 0.000,C 90.000,E1 53.290} C_DIS
LIN {X -0.010,Y -435.217,Z 651.093,A 0.000,B 0.000,C 90.000,E1 52.763} C_DIS
LIN {X -0.034,Y -435.210,Z 651.093,A 0.000,B 0.000,C 90.000,E1 52.763} C_DIS
LIN {X 0.097,Y -431.801,Z 651.083,A 0.000,B 0.000,C 90.000,E1 50.964} C_DIS
LIN {X 0.021,Y -431.089,Z 651.081,A 0.000,B 0.000,C 90.000,E1 50.642} C_DIS
LIN {X 0.018,Y -421.944,Z 651.059,A 0.000,B 0.000,C 90.000,E1 46.620} C_DIS
LIN {X -0.110,Y -421.128,Z 651.057,A 0.000,B 0.000,C 90.000,E1 46.215} C_DIS
LIN {X -0.228,Y -421.322,Z 651.044,A 0.000,B 0.000,C 90.000,E1 43.947} C_DIS
LIN {X 0.057,Y -421.834,Z 651.027,A 0.000,B 0.000,C 90.000,E1 40.862} C_DIS
LIN {X 0.087,Y -422.473,Z 651.016,A 0.000,B 0.000,C 90.000,E1 38.830} C_DIS
LIN {X -0.188,Y -423.535,Z 651.003,A 0.000,B 0.000,C 90.000,E1 36.503} C_DIS
LIN {X 0.020,Y -424.622,Z 650.991,A 0.000,B 0.000,C 90.000,E1 34.452} C_DIS
LIN {X 0.129,Y -425.581,Z 650.980,A 0.000,B 0.000,C 90.000,E1 32.418} C_DIS
LIN {X 0.036,Y -426.705,Z 650.967,A 0.000,B 0.000,C 90.000,E1 30.079} C_DIS
LIN {X -0.010,Y -427.392,Z 650.960,A 0.000,B 0.000,C 90.000,E1 28.743} C_DIS
LIN {X -0.097,Y -428.462,Z 650.949,A 0.000,B 0.000,C 90.000,E1 26.744} C_DIS
LIN {X -0.152,Y -429.410,Z 650.939,A 0.000,B 0.000,C 90.000,E1 25.079} C_DIS
LIN {X 0.036,Y -431.144,Z 650.926,A 0.000,B 0.000,C 90.000,E1 22.717} C_DIS
LIN {X 0.080,Y -432.534,Z 650.917,A 0.000,B 0.000,C 90.000,E1 21.046} C_DIS
LIN {X -0.008,Y -433.719,Z 650.908,A 0.000,B 0.000,C 90.000,E1 19.396} C_DIS
LIN {X -0.164,Y -435.096,Z 650.895,A 0.000,B 0.000,C 90.000,E1 17.094} C_DIS
LIN {X -0.125,Y -436.641,Z 650.882,A 0.000,B 0.000,C 90.000,E1 14.773} C_DIS
LIN {X 0.032,Y -438.263,Z 650.871,A 0.000,B 0.000,C 90.000,E1 12.771} C_DIS
LIN {X 0.009,Y -440.613,Z 650.856,A 0.000,B 0.000,C 90.000,E1 10.141} C_DIS
LIN {X -0.089,Y -443.282,Z 650.842,A 0.000,B 0.000,C 90.000,E1 7.530} C_DIS
LIN {X -0.195,Y -445.131,Z 650.833,A 0.000,B 0.000,C 90.000,E1 5.910} C_DIS
LIN {X -0.186,Y -448.733,Z 650.816,A 0.000,B 0.000,C 90.000,E1 2.980} C_DIS
LIN {X 0.000,Y -452.787,Z 650.800,A 0.000,B 0.000,C 90.000,E1 360.000} C_DIS
LIN {X -0.225,Y -457.202,Z 650.785,A 0.000,B 0.000,C 90.000,E1 357.249} C_DIS
LIN {X 0.037,Y -460.473,Z 650.774,A 0.000,B 0.000,C 90.000,E1 355.298} C_DIS
LIN {X 0.003,Y -463.885,Z 650.763,A 0.000,B 0.000,C 90.000,E1 353.394} C_DIS
LIN {X -0.140,Y -467.837,Z 650.751,A 0.000,B 0.000,C 90.000,E1 351.197} C_DIS
LIN {X 0.058,Y -471.126,Z 650.741,A 0.000,B 0.000,C 90.000,E1 349.285} C_DIS
LIN {X 0.040,Y -474.383,Z 650.730,A 0.000,B 0.000,C 90.000,E1 347.409} C_DIS
LIN {X 0.055,Y -478.418,Z 650.718,A 0.000,B 0.000,C 90.000,E1 345.227} C_DIS
LIN {X -0.001,Y -481.309,Z 650.709,A 0.000,B 0.000,C 90.000,E1 343.685} C_DIS
LIN {X 0.132,Y -484.910,Z 650.699,A 0.000,B 0.000,C 90.000,E1 341.819} C_DIS
LIN {X -0.115,Y -488.497,Z 650.689,A 0.000,B 0.000,C 90.000,E1 340.007} C_DIS
LIN {X -0.012,Y -490.961,Z 650.682,A 0.000,B 0.000,C 90.000,E1 338.773} C_DIS
LIN {X 0.134,Y -493.284,Z 650.675,A 0.000,B 0.000,C 90.000,E1 337.539} C_DIS
LIN {X -0.143,Y -495.470,Z 650.669,A 0.000,B 0.000,C 90.000,E1 336.357} C_DIS
LIN {X 0.265,Y -497.488,Z 650.662,A 0.000,B 0.000,C 90.000,E1 335.101} C_DIS
LIN {X -0.081,Y -500.491,Z 650.652,A 0.000,B 0.000,C 90.000,E1 333.332} C_DIS
LIN {X -0.055,Y -505.877,Z 650.635,A 0.000,B 0.000,C 90.000,E1 330.333} C_DIS
LIN {X 0.205,Y -508.088,Z 650.630,A 0.000,B 0.000,C 90.000,E1 329.410} C_DIS
LIN {X -0.278,Y -510.030,Z 650.627,A 0.000,B 0.000,C 90.000,E1 328.869} C_DIS
LIN {X 0.067,Y -511.260,Z 650.625,A 0.000,B 0.000,C 90.000,E1 328.535} C_DIS
LIN {X -0.212,Y -513.816,Z 650.623,A 0.000,B 0.000,C 90.000,E1 328.122} C_DIS
LIN {X 0.137,Y -516.025,Z 650.621,A 0.000,B 0.000,C 90.000,E1 327.788} C_DIS
LIN {X 0.171,Y -520.316,Z 650.619,A 0.000,B 0.000,C 90.000,E1 327.327} C_DIS
LIN {X 0.059,Y -524.100,Z 650.617,A 0.000,B 0.000,C 90.000,E1 326.993} C_DIS
LIN {X 0.103,Y -537.545,Z 650.611,A 0.000,B 0.000,C 90.000,E1 325.928} C_DIS
LIN {X 0.164,Y -547.730,Z 650.606,A 0.000,B 0.000,C 90.000,E1 325.102} C_DIS
LIN {X -0.096,Y -554.800,Z 650.603,A 0.000,B 0.000,C 90.000,E1 324.529} C_DIS
LIN {X -0.365,Y -564.537,Z 650.598,A 0.000,B 0.000,C 90.000,E1 323.703} C_DIS
LIN {X -0.030,Y -571.322,Z 650.595,A 0.000,B 0.000,C 90.000,E1 323.050} C_DIS
LIN {X 0.266,Y -579.329,Z 650.591,A 0.000,B 0.000,C 90.000,E1 322.271} C_DIS
LIN {X 0.025,Y -589.783,Z 650.585,A 0.000,B 0.000,C 90.000,E1 321.295} C_DIS
LIN {X 0.235,Y -600.073,Z 650.579,A 0.000,B 0.000,C 90.000,E1 320.275} C_DIS
LIN {X -0.119,Y -605.824,Z 650.576,A 0.000,B 0.000,C 90.000,E1 319.703} C_DIS
LIN {X 0.035,Y -609.430,Z 650.574,A 0.000,B 0.000,C 90.000,E1 319.299} C_DIS
LIN {X 0.155,Y -613.960,Z 650.571,A 0.000,B 0.000,C 90.000,E1 318.771} C_DIS
LIN {X -0.003,Y -617.134,Z 650.569,A 0.000,B 0.000,C 90.000,E1 318.405} C_DIS
LIN {X 0.054,Y -622.195,Z 650.565,A 0.000,B 0.000,C 90.000,E1 317.757} C_DIS
LIN {X 0.044,Y -628.728,Z 650.560,A 0.000,B 0.000,C 90.000,E1 316.863} C_DIS
LIN {X 0.304,Y -631.412,Z 650.558,A 0.000,B 0.000,C 90.000,E1 316.458} C_DIS
LIN {X -0.124,Y -638.274,Z 650.553,A 0.000,B 0.000,C 90.000,E1 315.486} C_DIS
LIN {X 0.026,Y -644.023,Z 650.548,A 0.000,B 0.000,C 90.000,E1 314.595} C_DIS
LIN {X -0.084,Y -650.916,Z 650.542,A 0.000,B 0.000,C 90.000,E1 313.500} C_DIS
LIN {X -0.011,Y -653.901,Z 650.539,A 0.000,B 0.000,C 90.000,E1 313.014} C_DIS
LIN {X -0.097,Y -656.798,Z 650.536,A 0.000,B 0.000,C 90.000,E1 312.528} C_DIS
LIN {X 0.295,Y -660.874,Z 650.532,A 0.000,B 0.000,C 90.000,E1 311.757} C_DIS
LIN {X -0.207,Y -664.807,Z 650.528,A 0.000,B 0.000,C 90.000,E1 311.067} C_DIS
LIN {X -0.204,Y -667.890,Z 650.525,A 0.000,B 0.000,C 90.000,E1 310.458} C_DIS
LIN {X -0.139,Y -671.276,Z 650.521,A 0.000,B 0.000,C 90.000,E1 309.725} C_DIS
LIN {X -0.036,Y -674.372,Z 650.517,A 0.000,B 0.000,C 90.000,E1 308.991} C_DIS
LIN {X 0.098,Y -677.215,Z 650.513,A 0.000,B 0.000,C 90.000,E1 308.257} C_DIS
LIN {X 0.261,Y -679.769,Z 650.509,A 0.000,B 0.000,C 90.000,E1 307.523} C_DIS
LIN {X 0.054,Y -682.908,Z 650.503,A 0.000,B 0.000,C 90.000,E1 306.583} C_DIS
LIN {X -0.141,Y -685.075,Z 650.499,A 0.000,B 0.000,C 90.000,E1 305.884} C_DIS
LIN {X -0.096,Y -688.533,Z 650.493,A 0.000,B 0.000,C 90.000,E1 304.692} C_DIS
LIN {X 0.358,Y -691.023,Z 650.487,A 0.000,B 0.000,C 90.000,E1 303.706} C_DIS
LIN {X 0.105,Y -693.938,Z 650.481,A 0.000,B 0.000,C 90.000,E1 302.546} C_DIS
LIN {X -0.108,Y -696.584,Z 650.474,A 0.000,B 0.000,C 90.000,E1 301.386} C_DIS
LIN {X 0.043,Y -698.005,Z 650.470,A 0.000,B 0.000,C 90.000,E1 300.669} C_DIS
LIN {X 0.139,Y -700.147,Z 650.464,A 0.000,B 0.000,C 90.000,E1 299.489} C_DIS
LIN {X -0.001,Y -701.699,Z 650.459,A 0.000,B 0.000,C 90.000,E1 298.565} C_DIS
LIN {X 0.149,Y -703.359,Z 650.452,A 0.000,B 0.000,C 90.000,E1 297.385} C_DIS
LIN {X -0.004,Y -704.774,Z 650.446,A 0.000,B 0.000,C 90.000,E1 296.232} C_DIS
LIN {X -0.081,Y -704.901,Z 650.442,A 0.000,B 0.000,C 90.000,E1 295.540} C_DIS
LIN {X -0.142,Y -704.157,Z 650.439,A 0.000,B 0.000,C 90.000,E1 295.079} C_DIS
LIN {X 0.143,Y -703.534,Z 650.438,A 0.000,B 0.000,C 90.000,E1 294.823} C_DIS
LIN {X -0.226,Y -700.696,Z 650.435,A 0.000,B 0.000,C 90.000,E1 294.387} C_DIS
LIN {X -0.089,Y -699.907,Z 650.435,A 0.000,B 0.000,C 90.000,E1 294.259} C_DIS
LIN {X 0.046,Y -698.819,Z 650.434,A 0.000,B 0.000,C 90.000,E1 294.131} C_DIS
LIN {X -0.105,Y -697.159,Z 650.433,A 0.000,B 0.000,C 90.000,E1 294.027} C_DIS
LIN {X -0.240,Y -691.327,Z 650.432,A 0.000,B 0.000,C 90.000,E1 293.770} C_DIS
LIN {X -0.200,Y -689.378,Z 650.432,A 0.000,B 0.000,C 90.000,E1 293.695} C_DIS
LIN {X 0.193,Y -686.969,Z 650.431,A 0.000,B 0.000,C 90.000,E1 293.590} C_DIS
LIN {X 0.004,Y -680.222,Z 650.430,A 0.000,B 0.000,C 90.000,E1 293.462} C_DIS
LIN {X 0.276,Y -670.501,Z 650.430,A 0.000,B 0.000,C 90.000,E1 293.334} C_DIS
LIN {X 0.018,Y -661.453,Z 650.429,A 0.000,B 0.000,C 90.000,E1 293.259} C_DIS
LIN {X -0.155,Y -651.284,Z 650.428,A 0.000,B 0.000,C 90.000,E1 293.131} C_DIS
LIN {X -0.045,Y -641.684,Z 650.428,A 0.000,B 0.000,C 90.000,E1 292.950} C_DIS
LIN {X 0.194,Y -631.487,Z 650.426,A 0.000,B 0.000,C 90.000,E1 292.717} C_DIS
LIN {X 0.178,Y -618.491,Z 650.424,A 0.000,B 0.000,C 90.000,E1 292.386} C_DIS
LIN {X 0.261,Y -597.994,Z 650.421,A 0.000,B 0.000,C 90.000,E1 291.770} C_DIS
LIN {X 0.161,Y -580.571,Z 650.418,A 0.000,B 0.000,C 90.000,E1 291.227} C_DIS
LIN {X -0.212,Y -573.103,Z 650.417,A 0.000,B 0.000,C 90.000,E1 291.046} C_DIS
LIN {X -0.152,Y -563.051,Z 650.415,A 0.000,B 0.000,C 90.000,E1 290.737} C_DIS
LIN {X 0.194,Y -559.718,Z 650.414,A 0.000,B 0.000,C 90.000,E1 290.556} C_DIS
LIN {X 0.010,Y -556.544,Z 650.413,A 0.000,B 0.000,C 90.000,E1 290.375} C_DIS
LIN {X -0.045,Y -556.502,Z 650.413,A 0.000,B 0.000,C 90.000,E1 290.375} C_DIS
LIN {X 0.070,Y -555.911,Z 650.413,A 0.000,B 0.000,C 90.000,E1 290.248} C_DIS
LIN {X -0.196,Y -555.570,Z 650.411,A 0.000,B 0.000,C 90.000,E1 290.066} C_DIS
LIN {X 0.093,Y -555.242,Z 650.410,A 0.000,B 0.000,C 90.000,E1 289.758} C_DIS
LIN {X -0.105,Y -555.032,Z 650.401,A 0.000,B 0.000,C 90.000,E1 288.109} C_DIS
LIN {X 0.259,Y -554.719,Z 650.393,A 0.000,B 0.000,C 90.000,E1 286.677} C_DIS
LIN {X -0.178,Y -554.343,Z 650.387,A 0.000,B 0.000,C 90.000,E1 285.607} C_DIS
LIN {X 0.039,Y -553.729,Z 650.379,A 0.000,B 0.000,C 90.000,E1 284.189} C_DIS
LIN {X 0.123,Y -553.115,Z 650.373,A 0.000,B 0.000,C 90.000,E1 283.063} C_DIS
LIN {X -0.108,Y -552.113,Z 650.362,A 0.000,B 0.000,C 90.000,E1 281.130} C_DIS
LIN {X 0.077,Y -551.308,Z 650.351,A 0.000,B 0.000,C 90.000,E1 279.151} C_DIS
LIN {X 0.154,Y -550.710,Z 650.340,A 0.000,B 0.000,C 90.000,E1 277.182} C_DIS
LIN {X 0.042,Y -550.292,Z 650.331,A 0.000,B 0.000,C 90.000,E1 275.511} C_DIS
LIN {X -0.172,Y -550.011,Z 650.323,A 0.000,B 0.000,C 90.000,E1 274.131} C_DIS
LIN {X 0.152,Y -549.724,Z 650.315,A 0.000,B 0.000,C 90.000,E1 272.694} C_DIS
LIN {X -0.115,Y -549.307,Z 650.307,A 0.000,B 0.000,C 90.000,E1 271.318} C_DIS
LIN {X 0.200,Y -548.554,Z 650.298,A 0.000,B 0.000,C 90.000,E1 269.599} C_DIS
LIN {X 0.009,Y -547.530,Z 650.287,A 0.000,B 0.000,C 90.000,E1 267.650} C_DIS
LIN {X 0.251,Y -546.803,Z 650.279,A 0.000,B 0.000,C 90.000,E1 266.216} C_DIS
LIN {X -0.065,Y -546.063,Z 650.273,A 0.000,B 0.000,C 90.000,E1 265.122} C_DIS
LIN {X 0.183,Y -545.012,Z 650.265,A 0.000,B 0.000,C 90.000,E1 263.685} C_DIS
LIN {X -0.159,Y -543.972,Z 650.259,A 0.000,B 0.000,C 90.000,E1 262.591} C_DIS
LIN {X 0.175,Y -542.402,Z 650.251,A 0.000,B 0.000,C 90.000,E1 261.141} C_DIS
LIN {X -0.201,Y -539.687,Z 650.235,A 0.000,B 0.000,C 90.000,E1 258.342} C_DIS
LIN {X -0.048,Y -537.728,Z 650.223,A 0.000,B 0.000,C 90.000,E1 256.047} C_DIS
LIN {X -0.079,Y -536.240,Z 650.213,A 0.000,B 0.000,C 90.000,E1 254.338} C_DIS
LIN {X 0.142,Y -534.575,Z 650.203,A 0.000,B 0.000,C 90.000,E1 252.598} C_DIS
LIN {X -0.180,Y -532.978,Z 650.194,A 0.000,B 0.000,C 90.000,E1 250.913} C_DIS
LIN {X -0.268,Y -531.998,Z 650.189,A 0.000,B 0.000,C 90.000,E1 250.061} C_DIS
LIN {X -0.176,Y -530.431,Z 650.183,A 0.000,B 0.000,C 90.000,E1 248.901} C_DIS
LIN {X 0.270,Y -528.345,Z 650.175,A 0.000,B 0.000,C 90.000,E1 247.411} C_DIS
LIN {X -0.192,Y -526.513,Z 650.168,A 0.000,B 0.000,C 90.000,E1 246.305} C_DIS
LIN {X -0.090,Y -523.898,Z 650.160,A 0.000,B 0.000,C 90.000,E1 244.845} C_DIS
LIN {X 0.288,Y -521.599,Z 650.154,A 0.000,B 0.000,C 90.000,E1 243.640} C_DIS
LIN {X 0.159,Y -519.207,Z 650.147,A 0.000,B 0.000,C 90.000,E1 242.487} C_DIS
LIN {X -0.098,Y -516.139,Z 650.139,A 0.000,B 0.000,C 90.000,E1 241.051} C_DIS
LIN {X 0.283,Y -514.209,Z 650.134,A 0.000,B 0.000,C 90.000,E1 240.127} C_DIS
LIN {X -0.170,Y -510.160,Z 650.124,A 0.000,B 0.000,C 90.000,E1 238.408} C_DIS
LIN {X -0.072,Y -506.750,Z 650.116,A 0.000,B 0.000,C 90.000,E1 236.914} C_DIS
LIN {X 0.039,Y -504.659,Z 650.111,A 0.000,B 0.000,C 90.000,E1 236.008} C_DIS
LIN {X 0.015,Y -501.561,Z 650.105,A 0.000,B 0.000,C 90.000,E1 234.815} C_DIS
LIN {X -0.177,Y -497.669,Z 650.096,A 0.000,B 0.000,C 90.000,E1 233.336} C_DIS
LIN {X 0.109,Y -491.702,Z 650.083,A 0.000,B 0.000,C 90.000,E1 230.884} C_DIS
LIN {X 0.078,Y -485.883,Z 650.069,A 0.000,B 0.000,C 90.000,E1 228.447} C_DIS
LIN {X -0.061,Y -481.501,Z 650.059,A 0.000,B 0.000,C 90.000,E1 226.620} C_DIS
LIN {X -0.230,Y -478.505,Z 650.052,A 0.000,B 0.000,C 90.000,E1 225.405} C_DIS
LIN {X 0.012,Y -474.845,Z 650.044,A 0.000,B 0.000,C 90.000,E1 223.824} C_DIS
LIN {X 0.043,Y -469.822,Z 650.031,A 0.000,B 0.000,C 90.000,E1 221.634} C_DIS
LIN {X -0.023,Y -465.051,Z 650.019,A 0.000,B 0.000,C 90.000,E1 219.439} C_DIS
LIN {X 0.096,Y -461.053,Z 650.009,A 0.000,B 0.000,C 90.000,E1 217.523} C_DIS
LIN {X -0.063,Y -456.633,Z 649.996,A 0.000,B 0.000,C 90.000,E1 215.311} C_DIS
LIN {X -0.047,Y -453.660,Z 649.987,A 0.000,B 0.000,C 90.000,E1 213.706} C_DIS
LIN {X -0.169,Y -449.541,Z 649.975,A 0.000,B 0.000,C 90.000,E1 211.465} C_DIS
LIN {X 0.069,Y -446.075,Z 649.964,A 0.000,B 0.000,C 90.000,E1 209.489} C_DIS
LIN {X 0.114,Y -443.725,Z 649.957,A 0.000,B 0.000,C 90.000,E1 208.180} C_DIS
LIN {X 0.000,Y -440.154,Z 649.946,A 0.000,B 0.000,C 90.000,E1 206.232} C_DIS
LIN {X 0.137,Y -437.777,Z 649.938,A 0.000,B 0.000,C 90.000,E1 204.899} C_DIS
LIN {X -0.111,Y -434.144,Z 649.927,A 0.000,B 0.000,C 90.000,E1 202.950} C_DIS
LIN {X -0.031,Y -431.207,Z 649.918,A 0.000,B 0.000,C 90.000,E1 201.280} C_DIS
LIN {X 0.042,Y -427.729,Z 649.907,A 0.000,B 0.000,C 90.000,E1 199.268} C_DIS
LIN {X -0.090,Y -425.465,Z 649.900,A 0.000,B 0.000,C 90.000,E1 197.946} C_DIS
LIN {X 0.112,Y -422.129,Z 649.888,A 0.000,B 0.000,C 90.000,E1 195.898} C_DIS
LIN {X -0.167,Y -419.448,Z 649.879,A 0.000,B 0.000,C 90.000,E1 194.245} C_DIS
LIN {X -0.143,Y -417.307,Z 649.872,A 0.000,B 0.000,C 90.000,E1 192.883} C_DIS
LIN {X -0.061,Y -413.119,Z 649.856,A 0.000,B 0.000,C 90.000,E1 190.141} C_DIS
LIN {X 0.164,Y -410.112,Z 649.845,A 0.000,B 0.000,C 90.000,E1 188.049} C_DIS
LIN {X -0.179,Y -406.157,Z 649.830,A 0.000,B 0.000,C 90.000,E1 185.334} C_DIS
LIN {X 0.049,Y -402.663,Z 649.814,A 0.000,B 0.000,C 90.000,E1 182.522} C_DIS
LIN {X 0.094,Y -399.456,Z 649.797,A 0.000,B 0.000,C 90.000,E1 179.370} C_DIS
LIN {X 0.040,Y -397.086,Z 649.779,A 0.000,B 0.000,C 90.000,E1 176.216} C_DIS
LIN {X 0.062,Y -395.709,Z 649.763,A 0.000,B 0.000,C 90.000,E1 173.394} C_DIS
LIN {X 0.083,Y -394.712,Z 649.744,A 0.000,B 0.000,C 90.000,E1 169.859} C_DIS
LIN {X -0.128,Y -394.416,Z 649.728,A 0.000,B 0.000,C 90.000,E1 167.061} C_DIS
LIN {X -0.106,Y -394.444,Z 649.716,A 0.000,B 0.000,C 90.000,E1 164.936} C_DIS
LIN {X 0.132,Y -394.662,Z 649.704,A 0.000,B 0.000,C 90.000,E1 162.779} C_DIS
LIN {X 0.000,Y -395.013,Z 649.693,A 0.000,B 0.000,C 90.000,E1 160.678} C_DIS
LIN {X 0.130,Y -395.396,Z 649.681,A 0.000,B 0.000,C 90.000,E1 158.539} C_DIS
LIN {X -0.010,Y -395.791,Z 649.671,A 0.000,B 0.000,C 90.000,E1 156.794} C_DIS
LIN {X -0.142,Y -396.201,Z 649.661,A 0.000,B 0.000,C 90.000,E1 155.049} C_DIS
LIN {X 0.068,Y -396.653,Z 649.652,A 0.000,B 0.000,C 90.000,E1 153.256} C_DIS
LIN {X -0.064,Y -397.063,Z 649.642,A 0.000,B 0.000,C 90.000,E1 151.513} C_DIS
LIN {X -0.125,Y -397.616,Z 649.630,A 0.000,B 0.000,C 90.000,E1 149.410} C_DIS
LIN {X 0.233,Y -398.244,Z 649.618,A 0.000,B 0.000,C 90.000,E1 147.248} C_DIS
LIN {X -0.059,Y -399.022,Z 649.607,A 0.000,B 0.000,C 90.000,E1 145.182} C_DIS
LIN {X 0.127,Y -399.954,Z 649.595,A 0.000,B 0.000,C 90.000,E1 143.050} C_DIS
LIN {X 0.028,Y -400.605,Z 649.587,A 0.000,B 0.000,C 90.000,E1 141.662} C_DIS
LIN {X 0.177,Y -401.564,Z 649.575,A 0.000,B 0.000,C 90.000,E1 139.542} C_DIS
LIN {X -0.129,Y -402.433,Z 649.566,A 0.000,B 0.000,C 90.000,E1 137.838} C_DIS
LIN {X -0.019,Y -403.445,Z 649.554,A 0.000,B 0.000,C 90.000,E1 135.729} C_DIS
LIN {X 0.271,Y -404.313,Z 649.544,A 0.000,B 0.000,C 90.000,E1 133.947} C_DIS
LIN {X -0.147,Y -405.638,Z 649.533,A 0.000,B 0.000,C 90.000,E1 131.919} C_DIS
LIN {X -0.179,Y -406.311,Z 649.529,A 0.000,B 0.000,C 90.000,E1 131.229} C_DIS
LIN {X -0.207,Y -407.354,Z 649.525,A 0.000,B 0.000,C 90.000,E1 130.539} C_DIS
LIN {X 0.020,Y -407.596,Z 649.524,A 0.000,B 0.000,C 90.000,E1 130.334} C_DIS
LIN {X -0.099,Y -409.741,Z 649.520,A 0.000,B 0.000,C 90.000,E1 129.564} C_DIS
LIN {X -0.026,Y -411.564,Z 649.518,A 0.000,B 0.000,C 90.000,E1 129.197} C_DIS
LIN {X -0.107,Y -412.795,Z 649.517,A 0.000,B 0.000,C 90.000,E1 129.036} C_DIS
LIN {X 0.169,Y -415.764,Z 649.515,A 0.000,B 0.000,C 90.000,E1 128.669} C_DIS
LIN {X 0.068,Y -419.143,Z 649.513,A 0.000,B 0.000,C 90.000,E1 128.382} C_DIS
LIN {X -0.036,Y -426.894,Z 649.510,A 0.000,B 0.000,C 90.000,E1 127.810} C_DIS
LIN {X -0.067,Y -448.306,Z 649.502,A 0.000,B 0.000,C 90.000,E1 126.377} C_DIS
LIN {X -0.103,Y -457.956,Z 649.498,A 0.000,B 0.000,C 90.000,E1 125.724} C_DIS
LIN {X -0.102,Y -468.863,Z 649.494,A 0.000,B 0.000,C 90.000,E1 124.945} C_DIS
LIN {X -0.002,Y -477.697,Z 649.490,A 0.000,B 0.000,C 90.000,E1 124.278} C_DIS
LIN {X -0.205,Y -485.344,Z 649.487,A 0.000,B 0.000,C 90.000,E1 123.706} C_DIS
LIN {X 0.264,Y -493.848,Z 649.483,A 0.000,B 0.000,C 90.000,E1 122.959} C_DIS
LIN {X 0.017,Y -499.482,Z 649.481,A 0.000,B 0.000,C 90.000,E1 122.498} C_DIS
LIN {X 0.004,Y -509.626,Z 649.476,A 0.000,B 0.000,C 90.000,E1 121.592} C_DIS
LIN {X 0.213,Y -519.290,Z 649.471,A 0.000,B 0.000,C 90.000,E1 120.669} C_DIS
LIN {X 0.069,Y -527.257,Z 649.466,A 0.000,B 0.000,C 90.000,E1 119.873} C_DIS
LIN {X -0.109,Y -529.926,Z 649.465,A 0.000,B 0.000,C 90.000,E1 119.617} C_DIS
LIN {X -0.238,Y -534.818,Z 649.461,A 0.000,B 0.000,C 90.000,E1 119.077} C_DIS
LIN {X -0.060,Y -539.459,Z 649.458,A 0.000,B 0.000,C 90.000,E1 118.487} C_DIS
LIN {X 0.264,Y -542.692,Z 649.456,A 0.000,B 0.000,C 90.000,E1 118.025} C_DIS
LIN {X -0.038,Y -547.302,Z 649.452,A 0.000,B 0.000,C 90.000,E1 117.385} C_DIS
LIN {X -0.286,Y -549.004,Z 649.451,A 0.000,B 0.000,C 90.000,E1 117.129} C_DIS
LIN {X -0.024,Y -552.234,Z 649.447,A 0.000,B 0.000,C 90.000,E1 116.539} C_DIS
LIN {X -0.096,Y -555.943,Z 649.444,A 0.000,B 0.000,C 90.000,E1 115.848} C_DIS
LIN {X 0.125,Y -560.972,Z 649.437,A 0.000,B 0.000,C 90.000,E1 114.719} C_DIS
LIN {X 0.037,Y -564.411,Z 649.433,A 0.000,B 0.000,C 90.000,E1 113.898} C_DIS
LIN {X -0.207,Y -568.738,Z 649.427,A 0.000,B 0.000,C 90.000,E1 112.823} C_DIS
LIN {X 0.084,Y -571.629,Z 649.422,A 0.000,B 0.000,C 90.000,E1 111.972} C_DIS
LIN {X 0.091,Y -574.207,Z 649.418,A 0.000,B 0.000,C 90.000,E1 111.153} C_DIS
LIN {X 0.084,Y -577.294,Z 649.412,A 0.000,B 0.000,C 90.000,E1 110.066} C_DIS
LIN {X 0.320,Y -580.032,Z 649.406,A 0.000,B 0.000,C 90.000,E1 108.960} C_DIS
LIN {X -0.154,Y -582.487,Z 649.400,A 0.000,B 0.000,C 90.000,E1 107.928} C_DIS
LIN {X 0.084,Y -586.524,Z 649.389,A 0.000,B 0.000,C 90.000,E1 106.024} C_DIS
LIN {X -0.139,Y -590.718,Z 649.379,A 0.000,B 0.000,C 90.000,E1 104.175} C_DIS
LIN {X 0.044,Y -593.708,Z 649.371,A 0.000,B 0.000,C 90.000,E1 102.827} C_DIS
LIN {X 0.002,Y -596.012,Z 649.365,A 0.000,B 0.000,C 90.000,E1 101.771} C_DIS
LIN {X -0.121,Y -599.434,Z 649.357,A 0.000,B 0.000,C 90.000,E1 100.197} C_DIS
LIN {X 0.109,Y -602.214,Z 649.349,A 0.000,B 0.000,C 90.000,E1 98.859} C_DIS
LIN {X -0.302,Y -604.811,Z 649.342,A 0.000,B 0.000,C 90.000,E1 97.587} C_DIS
LIN {X 0.283,Y -606.651,Z 649.336,A 0.000,B 0.000,C 90.000,E1 96.486} C_DIS
LIN {X -0.103,Y -607.997,Z 649.332,A 0.000,B 0.000,C 90.000,E1 95.739} C_DIS
LIN {X 0.116,Y -610.010,Z 649.325,A 0.000,B 0.000,C 90.000,E1 94.416} C_DIS
LIN {X -0.246,Y -611.872,Z 649.317,A 0.000,B 0.000,C 90.000,E1 93.151} C_DIS
LIN {X -0.028,Y -613.385,Z 649.310,A 0.000,B 0.000,C 90.000,E1 91.835} C_DIS
LIN {X 0.260,Y -614.149,Z 649.306,A 0.000,B 0.000,C 90.000,E1 91.031} C_DIS
LIN {X -0.086,Y -615.148,Z 649.299,A 0.000,B 0.000,C 90.000,E1 89.771} C_DIS
END
